Yaskawa INFORM job: DEMO_ROOF_SIDE_0625_3PAINT_16.JBI

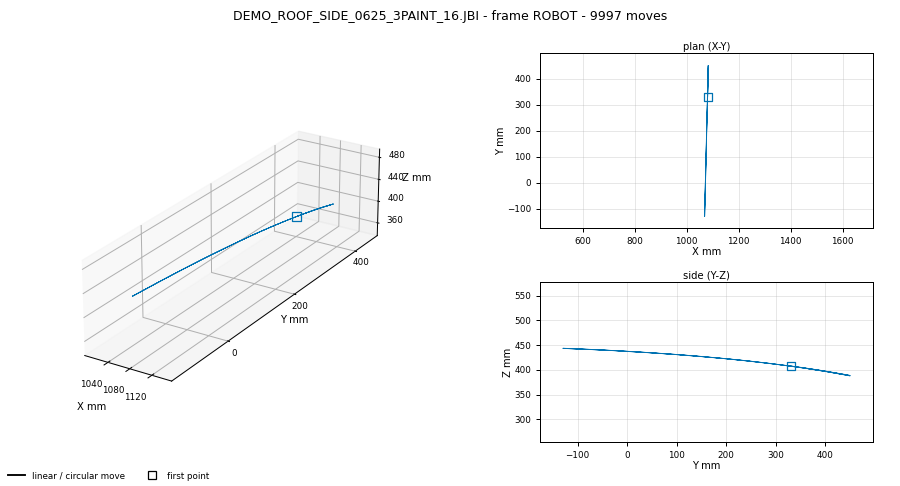
[picture p0: tool path of DEMO_ROOF_SIDE_0625_3PAINT_16.JBI in frame ROBOT, 9997 of 9997 moves have a stored position in this frame; points joined in program order, loops and branches not executed]
/JOB
//NAME DEMO_ROOF_SIDE_0625_3PAINT16
//POS
///NPOS 9997,0,0,0,0,0
///TOOL 0
///USER 0
///POSTYPE ROBOT
///RECTAN
///RCONF 1,0,0,0,0,0,0,0,0,0,0,0,0,0,0,0,0,0,0,0,0,0,0,0
C00000=1080.812,330.595,407.763,175.918,27.097,154.616
C00001=1080.821,331.010,407.707,175.923,27.105,154.617
C00002=1080.832,331.424,407.651,175.928,27.113,154.618
C00003=1080.838,331.672,407.618,175.931,27.117,154.619
C00004=1080.844,331.919,407.584,175.934,27.122,154.620
C00005=1080.849,332.167,407.551,175.937,27.126,154.620
C00006=1080.856,332.416,407.518,175.940,27.131,154.621
C00007=1080.862,332.663,407.484,175.943,27.136,154.622
C00008=1080.868,332.911,407.450,175.947,27.141,154.623
C00009=1080.873,333.158,407.416,175.950,27.146,154.623
C00010=1080.879,333.406,407.383,175.953,27.150,154.624
C00011=1080.885,333.653,407.349,175.956,27.155,154.625
C00012=1080.892,333.902,407.316,175.959,27.160,154.626
C00013=1080.898,334.149,407.282,175.962,27.165,154.627
C00014=1080.904,334.396,407.248,175.965,27.170,154.627
C00015=1080.909,334.644,407.214,175.968,27.174,154.628
C00016=1080.915,334.891,407.180,175.971,27.179,154.629
C00017=1080.921,335.140,407.147,175.975,27.183,154.630
C00018=1080.927,335.387,407.112,175.978,27.188,154.630
C00019=1080.933,335.635,407.078,175.981,27.193,154.631
C00020=1080.939,335.883,407.045,175.984,27.198,154.632
C00021=1080.946,336.130,407.011,175.987,27.202,154.633
C00022=1080.951,336.377,406.977,175.990,27.207,154.633
C00023=1080.957,336.625,406.944,175.994,27.212,154.634
C00024=1080.963,336.873,406.909,175.997,27.217,154.635
C00025=1080.969,337.121,406.875,176.000,27.222,154.636
C00026=1080.975,337.368,406.841,176.003,27.227,154.637
C00027=1080.981,337.616,406.808,176.006,27.232,154.637
C00028=1080.987,337.864,406.774,176.009,27.236,154.638
C00029=1080.993,338.111,406.740,176.012,27.241,154.639
C00030=1080.999,338.359,406.705,176.015,27.246,154.640
C00031=1081.005,338.606,406.671,176.018,27.251,154.641
C00032=1081.011,338.854,406.637,176.022,27.256,154.642
C00033=1081.018,339.102,406.603,176.025,27.261,154.642
C00034=1081.024,339.349,406.569,176.028,27.266,154.643
C00035=1081.029,339.596,406.534,176.031,27.270,154.644
C00036=1081.035,339.845,406.500,176.034,27.276,154.645
C00037=1081.041,340.092,406.466,176.037,27.280,154.646
C00038=1081.047,340.340,406.432,176.040,27.285,154.646
C00039=1081.053,340.588,406.398,176.043,27.290,154.647
C00040=1081.059,340.835,406.364,176.047,27.295,154.648
C00041=1081.065,341.082,406.329,176.050,27.300,154.649
C00042=1081.071,341.330,406.294,176.053,27.305,154.650
C00043=1081.077,341.577,406.260,176.056,27.310,154.650
C00044=1081.083,341.825,406.225,176.059,27.315,154.651
C00045=1081.089,342.072,406.191,176.062,27.320,154.652
C00046=1081.095,342.320,406.157,176.065,27.325,154.653
C00047=1081.101,342.568,406.123,176.069,27.330,154.654
C00048=1081.106,342.815,406.088,176.072,27.335,154.655
C00049=1081.113,343.063,406.054,176.075,27.340,154.655
C00050=1081.119,343.310,406.019,176.078,27.345,154.656
C00051=1081.129,343.719,405.962,176.084,27.353,154.658
C00052=1081.140,344.129,405.905,176.089,27.362,154.659
C00053=1081.149,344.538,405.848,176.095,27.370,154.660
C00054=1081.159,344.947,405.790,176.100,27.379,154.662
C00055=1081.165,345.194,405.756,176.103,27.383,154.663
C00056=1081.171,345.442,405.720,176.106,27.389,154.664
C00057=1081.177,345.689,405.686,176.109,27.394,154.665
C00058=1081.183,345.937,405.651,176.113,27.399,154.665
C00059=1081.189,346.184,405.617,176.116,27.404,154.666
C00060=1081.195,346.432,405.582,176.119,27.409,154.667
C00061=1081.201,346.679,405.547,176.122,27.414,154.668
C00062=1081.207,346.927,405.512,176.125,27.419,154.669
C00063=1081.213,347.174,405.477,176.129,27.425,154.670
C00064=1081.219,347.422,405.443,176.132,27.430,154.671
C00065=1081.225,347.669,405.407,176.135,27.435,154.671
C00066=1081.231,347.917,405.373,176.138,27.440,154.672
C00067=1081.237,348.164,405.337,176.142,27.446,154.673
C00068=1081.243,348.412,405.303,176.145,27.451,154.674
C00069=1081.250,348.659,405.268,176.148,27.456,154.675
C00070=1081.255,348.906,405.233,176.151,27.461,154.676
C00071=1081.261,349.154,405.198,176.154,27.466,154.677
C00072=1081.267,349.401,405.163,176.158,27.472,154.678
C00073=1081.273,349.649,405.127,176.161,27.477,154.679
C00074=1081.280,349.897,405.093,176.164,27.482,154.680
C00075=1081.285,350.144,405.057,176.167,27.488,154.680
C00076=1081.292,350.391,405.022,176.171,27.493,154.681
C00077=1081.298,350.639,404.987,176.174,27.498,154.682
C00078=1081.304,350.886,404.952,176.177,27.504,154.683
C00079=1081.310,351.134,404.917,176.181,27.509,154.684
C00080=1081.317,351.381,404.882,176.184,27.514,154.685
C00081=1081.322,351.628,404.846,176.187,27.519,154.686
C00082=1081.328,351.876,404.811,176.190,27.525,154.687
C00083=1081.334,352.124,404.776,176.194,27.530,154.688
C00084=1081.340,352.371,404.741,176.197,27.535,154.689
C00085=1081.347,352.618,404.706,176.200,27.541,154.689
C00086=1081.353,352.866,404.670,176.203,27.546,154.690
C00087=1081.359,353.113,404.634,176.207,27.552,154.691
C00088=1081.364,353.360,404.599,176.210,27.557,154.692
C00089=1081.371,353.608,404.564,176.213,27.562,154.693
C00090=1081.377,353.855,404.528,176.217,27.568,154.694
C00091=1081.382,354.102,404.492,176.220,27.573,154.695
C00092=1081.388,354.350,404.457,176.223,27.579,154.696
C00093=1081.395,354.597,404.422,176.227,27.584,154.697
C00094=1081.401,354.845,404.386,176.229,27.590,154.698
C00095=1081.407,355.092,404.350,176.232,27.595,154.699
C00096=1081.413,355.340,404.315,176.236,27.601,154.700
C00097=1081.419,355.587,404.279,176.239,27.606,154.701
C00098=1081.425,355.835,404.244,176.242,27.612,154.702
C00099=1081.431,356.081,404.208,176.246,27.617,154.703
C00100=1081.437,356.329,404.172,176.249,27.622,154.704
C00101=1081.443,356.576,404.136,176.252,27.628,154.705
C00102=1081.449,356.824,404.101,176.256,27.634,154.706
C00103=1081.459,357.236,404.041,176.261,27.643,154.707
C00104=1081.470,357.647,403.981,176.267,27.652,154.709
C00105=1081.480,358.060,403.922,176.272,27.661,154.711
C00106=1081.490,358.472,403.862,176.278,27.671,154.712
C00107=1081.496,358.720,403.826,176.281,27.676,154.713
C00108=1081.503,358.967,403.790,176.284,27.682,154.714
C00109=1081.509,359.214,403.755,176.288,27.688,154.715
C00110=1081.515,359.461,403.719,176.291,27.693,154.716
C00111=1081.521,359.708,403.683,176.294,27.699,154.717
C00112=1081.527,359.955,403.647,176.298,27.705,154.718
C00113=1081.533,360.203,403.611,176.301,27.711,154.719
C00114=1081.540,360.450,403.574,176.305,27.717,154.720
C00115=1081.546,360.698,403.539,176.308,27.722,154.721
C00116=1081.552,360.945,403.502,176.311,27.727,154.722
C00117=1081.558,361.193,403.467,176.315,27.733,154.723
C00118=1081.564,361.440,403.430,176.318,27.739,154.724
C00119=1081.570,361.688,403.394,176.322,27.745,154.725
C00120=1081.576,361.935,403.357,176.324,27.751,154.726
C00121=1081.582,362.181,403.321,176.327,27.756,154.727
C00122=1081.588,362.429,403.286,176.331,27.762,154.728
C00123=1081.594,362.676,403.249,176.334,27.768,154.729
C00124=1081.601,362.923,403.213,176.338,27.774,154.730
C00125=1081.607,363.170,403.177,176.341,27.780,154.731
C00126=1081.613,363.417,403.140,176.344,27.785,154.733
C00127=1081.619,363.665,403.104,176.348,27.792,154.734
C00128=1081.626,363.912,403.068,176.351,27.797,154.735
C00129=1081.631,364.160,403.031,176.355,27.803,154.736
C00130=1081.637,364.407,402.995,176.358,27.809,154.737
C00131=1081.644,364.654,402.958,176.362,27.815,154.738
C00132=1081.650,364.901,402.922,176.365,27.821,154.739
C00133=1081.657,365.148,402.885,176.369,27.827,154.740
C00134=1081.663,365.396,402.849,176.372,27.833,154.741
C00135=1081.669,365.643,402.812,176.374,27.839,154.742
C00136=1081.675,365.891,402.776,176.378,27.845,154.743
C00137=1081.681,366.138,402.739,176.381,27.850,154.744
C00138=1081.687,366.385,402.702,176.385,27.857,154.745
C00139=1081.693,366.632,402.666,176.388,27.862,154.746
C00140=1081.699,366.879,402.629,176.392,27.869,154.748
C00141=1081.705,367.126,402.592,176.395,27.875,154.749
C00142=1081.712,367.373,402.555,176.399,27.881,154.750
C00143=1081.717,367.620,402.518,176.402,27.887,154.751
C00144=1081.724,367.867,402.482,176.406,27.893,154.752
C00145=1081.730,368.114,402.445,176.409,27.899,154.753
C00146=1081.736,368.362,402.408,176.412,27.906,154.754
C00147=1081.742,368.609,402.372,176.415,27.911,154.755
C00148=1081.748,368.857,402.334,176.419,27.918,154.756
C00149=1081.755,369.103,402.297,176.422,27.924,154.758
C00150=1081.761,369.350,402.261,176.426,27.930,154.759
C00151=1081.767,369.598,402.224,176.429,27.936,154.760
C00152=1081.773,369.845,402.187,176.433,27.942,154.761
C00153=1081.779,370.092,402.150,176.436,27.948,154.762
C00154=1081.786,370.339,402.113,176.440,27.955,154.763
C00155=1081.791,370.553,402.081,176.443,27.960,154.764
C00156=1081.796,370.767,402.050,176.446,27.966,154.765
C00157=1081.801,370.981,402.017,176.448,27.970,154.766
C00158=1081.807,371.195,401.985,176.451,27.976,154.767
C00159=1081.812,371.409,401.953,176.454,27.981,154.768
C00160=1081.818,371.623,401.920,176.457,27.987,154.769
C00161=1081.823,371.837,401.888,176.460,27.992,154.770
C00162=1081.828,372.052,401.856,176.463,27.998,154.771
C00163=1081.835,372.299,401.819,176.467,28.004,154.772
C00164=1081.841,372.546,401.782,176.470,28.010,154.773
C00165=1081.847,372.792,401.745,176.474,28.016,154.775
C00166=1081.854,373.041,401.707,176.477,28.023,154.776
C00167=1081.860,373.287,401.670,176.480,28.030,154.777
C00168=1081.866,373.534,401.633,176.483,28.036,154.778
C00169=1081.873,373.781,401.596,176.487,28.042,154.779
C00170=1081.879,374.028,401.558,176.491,28.048,154.781
C00171=1081.885,374.276,401.521,176.494,28.055,154.782
C00172=1081.891,374.522,401.484,176.498,28.061,154.783
C00173=1081.898,374.769,401.445,176.501,28.068,154.784
C00174=1081.903,375.017,401.408,176.505,28.074,154.785
C00175=1081.909,375.264,401.371,176.508,28.081,154.787
C00176=1081.916,375.510,401.333,176.511,28.087,154.788
C00177=1081.922,375.757,401.295,176.515,28.094,154.789
C00178=1081.928,376.005,401.258,176.518,28.100,154.790
C00179=1081.934,376.252,401.221,176.522,28.107,154.792
C00180=1081.941,376.499,401.183,176.526,28.114,154.793
C00181=1081.947,376.745,401.145,176.529,28.120,154.794
C00182=1081.953,376.992,401.108,176.533,28.127,154.795
C00183=1081.960,377.240,401.069,176.535,28.133,154.797
C00184=1081.965,377.487,401.032,176.539,28.140,154.798
C00185=1081.972,377.733,400.995,176.543,28.146,154.799
C00186=1081.978,377.981,400.957,176.546,28.153,154.800
C00187=1081.984,378.228,400.919,176.550,28.160,154.802
C00188=1081.991,378.475,400.881,176.554,28.167,154.803
C00189=1081.997,378.722,400.843,176.557,28.173,154.804
C00190=1082.004,378.969,400.806,176.560,28.180,154.805
C00191=1082.010,379.216,400.768,176.564,28.187,154.807
C00192=1082.016,379.462,400.730,176.567,28.193,154.808
C00193=1082.022,379.709,400.692,176.571,28.200,154.809
C00194=1082.028,379.956,400.654,176.575,28.207,154.810
C00195=1082.035,380.203,400.616,176.578,28.214,154.812
C00196=1082.041,380.450,400.578,176.582,28.220,154.813
C00197=1082.048,380.697,400.540,176.585,28.227,154.814
C00198=1082.054,380.944,400.503,176.588,28.234,154.816
C00199=1082.061,381.191,400.464,176.592,28.241,154.817
C00200=1082.067,381.438,400.426,176.596,28.248,154.818
C00201=1082.073,381.685,400.388,176.599,28.255,154.820
C00202=1082.080,381.932,400.350,176.603,28.261,154.821
C00203=1082.086,382.179,400.311,176.606,28.268,154.822
C00204=1082.092,382.426,400.273,176.610,28.275,154.823
C00205=1082.098,382.673,400.235,176.613,28.282,154.825
C00206=1082.105,382.920,400.197,176.617,28.289,154.826
C00207=1082.111,383.166,400.159,176.621,28.296,154.827
C00208=1082.118,383.413,400.120,176.624,28.303,154.829
C00209=1082.123,383.660,400.082,176.627,28.310,154.830
C00210=1082.130,383.907,400.043,176.631,28.318,154.832
C00211=1082.136,384.135,400.007,176.634,28.324,154.833
C00212=1082.141,384.364,399.972,176.638,28.330,154.834
C00213=1082.148,384.592,399.937,176.641,28.337,154.835
C00214=1082.153,384.819,399.901,176.644,28.344,154.837
C00215=1082.159,385.048,399.865,176.648,28.350,154.838
C00216=1082.165,385.276,399.830,176.651,28.356,154.839
C00217=1082.171,385.505,399.794,176.655,28.363,154.840
C00218=1082.177,385.733,399.759,176.658,28.370,154.842
C00219=1082.182,385.980,399.720,176.661,28.377,154.843
C00220=1082.189,386.227,399.681,176.665,28.385,154.844
C00221=1082.195,386.474,399.643,176.668,28.392,154.846
C00222=1082.201,386.721,399.605,176.672,28.399,154.847
C00223=1082.208,386.967,399.566,176.676,28.406,154.849
C00224=1082.214,387.214,399.527,176.680,28.413,154.850
C00225=1082.220,387.461,399.488,176.683,28.421,154.852
C00226=1082.227,387.708,399.450,176.686,28.428,154.853
C00227=1082.234,387.955,399.411,176.690,28.435,154.854
C00228=1082.240,388.202,399.372,176.694,28.442,154.856
C00229=1082.246,388.448,399.333,176.698,28.450,154.857
C00230=1082.253,388.695,399.294,176.701,28.458,154.859
C00231=1082.260,388.942,399.256,176.705,28.465,154.860
C00232=1082.266,389.189,399.216,176.708,28.472,154.862
C00233=1082.272,389.435,399.178,176.712,28.479,154.863
C00234=1082.279,389.682,399.139,176.716,28.487,154.865
C00235=1082.285,389.929,399.099,176.719,28.494,154.866
C00236=1082.292,390.176,399.061,176.723,28.502,154.867
C00237=1082.298,390.423,399.022,176.727,28.509,154.869
C00238=1082.304,390.669,398.983,176.731,28.517,154.870
C00239=1082.311,390.916,398.944,176.734,28.524,154.872
C00240=1082.318,391.163,398.905,176.738,28.531,154.873
C00241=1082.324,391.410,398.866,176.741,28.539,154.875
C00242=1082.330,391.657,398.827,176.745,28.546,154.876
C00243=1082.338,391.903,398.787,176.749,28.554,154.878
C00244=1082.344,392.150,398.748,176.753,28.562,154.879
C00245=1082.350,392.396,398.709,176.756,28.570,154.881
C00246=1082.356,392.643,398.670,176.760,28.578,154.882
C00247=1082.362,392.890,398.630,176.763,28.585,154.884
C00248=1082.369,393.137,398.591,176.767,28.593,154.885
C00249=1082.375,393.384,398.551,176.771,28.601,154.887
C00250=1082.382,393.630,398.512,176.774,28.608,154.888
C00251=1082.388,393.877,398.472,176.778,28.616,154.890
C00252=1082.395,394.124,398.434,176.782,28.624,154.892
C00253=1082.402,394.370,398.393,176.786,28.632,154.893
C00254=1082.408,394.618,398.354,176.790,28.639,154.895
C00255=1082.415,394.864,398.314,176.793,28.647,154.896
C00256=1082.421,395.111,398.275,176.797,28.655,154.898
C00257=1082.427,395.357,398.235,176.801,28.663,154.899
C00258=1082.434,395.604,398.196,176.805,28.671,154.901
C00259=1082.440,395.851,398.156,176.808,28.679,154.903
C00260=1082.446,396.098,398.116,176.812,28.687,154.904
C00261=1082.453,396.344,398.076,176.816,28.695,154.906
C00262=1082.460,396.591,398.037,176.819,28.703,154.907
C00263=1082.466,396.838,397.997,176.823,28.711,154.909
C00264=1082.472,397.084,397.957,176.826,28.719,154.911
C00265=1082.479,397.331,397.918,176.830,28.727,154.912
C00266=1082.486,397.578,397.878,176.834,28.735,154.914
C00267=1082.491,397.813,397.839,176.838,28.743,154.915
C00268=1082.498,398.048,397.802,176.842,28.750,154.917
C00269=1082.504,398.283,397.764,176.845,28.759,154.919
C00270=1082.510,398.519,397.725,176.848,28.766,154.920
C00271=1082.517,398.754,397.687,176.852,28.774,154.922
C00272=1082.523,398.989,397.650,176.856,28.782,154.923
C00273=1082.529,399.224,397.611,176.860,28.790,154.925
C00274=1082.536,399.461,397.573,176.863,28.798,154.926
C00275=1082.542,399.707,397.533,176.867,28.806,154.928
C00276=1082.548,399.954,397.493,176.871,28.814,154.930
C00277=1082.555,400.200,397.453,176.875,28.823,154.932
C00278=1082.561,400.447,397.413,176.878,28.831,154.933
C00279=1082.568,400.693,397.372,176.882,28.840,154.935
C00280=1082.575,400.940,397.332,176.886,28.848,154.937
C00281=1082.581,401.187,397.292,176.890,28.856,154.938
C00282=1082.587,401.433,397.252,176.893,28.865,154.940
C00283=1082.594,401.680,397.211,176.897,28.873,154.942
C00284=1082.601,401.927,397.171,176.901,28.882,154.944
C00285=1082.607,402.174,397.131,176.905,28.890,154.945
C00286=1082.614,402.420,397.090,176.908,28.898,154.947
C00287=1082.621,402.667,397.049,176.913,28.907,154.949
C00288=1082.627,402.913,397.009,176.917,28.916,154.950
C00289=1082.633,403.160,396.969,176.921,28.924,154.952
C00290=1082.641,403.406,396.928,176.924,28.933,154.954
C00291=1082.646,403.653,396.887,176.928,28.942,154.956
C00292=1082.653,403.900,396.847,176.932,28.950,154.958
C00293=1082.660,404.147,396.807,176.936,28.959,154.959
C00294=1082.666,404.393,396.766,176.939,28.968,154.961
C00295=1082.673,404.639,396.726,176.944,28.976,154.963
C00296=1082.680,404.886,396.684,176.948,28.985,154.965
C00297=1082.686,405.133,396.644,176.952,28.994,154.967
C00298=1082.692,405.379,396.603,176.955,29.002,154.968
C00299=1082.699,405.626,396.562,176.959,29.012,154.970
C00300=1082.706,405.872,396.522,176.964,29.021,154.972
C00301=1082.712,406.119,396.480,176.968,29.030,154.974
C00302=1082.719,406.365,396.439,176.971,29.038,154.976
C00303=1082.726,406.612,396.399,176.975,29.047,154.978
C00304=1082.733,406.858,396.358,176.979,29.056,154.980
C00305=1082.738,407.105,396.317,176.983,29.065,154.981
C00306=1082.746,407.352,396.276,176.987,29.074,154.983
C00307=1082.752,407.598,396.235,176.991,29.083,154.985
C00308=1082.759,407.845,396.193,176.995,29.092,154.987
C00309=1082.765,408.091,396.153,176.999,29.102,154.989
C00310=1082.772,408.338,396.111,177.003,29.111,154.991
C00311=1082.778,408.584,396.070,177.007,29.120,154.993
C00312=1082.785,408.831,396.029,177.011,29.129,154.995
C00313=1082.791,409.077,395.988,177.015,29.139,154.997
C00314=1082.798,409.324,395.947,177.019,29.148,154.999
C00315=1082.805,409.570,395.906,177.023,29.157,155.001
C00316=1082.811,409.817,395.864,177.027,29.167,155.003
C00317=1082.818,410.064,395.823,177.031,29.176,155.004
C00318=1082.824,410.310,395.781,177.035,29.185,155.006
C00319=1082.832,410.556,395.740,177.040,29.195,155.008
C00320=1082.838,410.803,395.699,177.043,29.204,155.010
C00321=1082.845,411.049,395.657,177.047,29.213,155.012
C00322=1082.851,411.296,395.616,177.052,29.223,155.014
C00323=1082.858,411.532,395.576,177.056,29.232,155.016
C00324=1082.864,411.768,395.536,177.059,29.241,155.018
C00325=1082.871,412.005,395.496,177.063,29.250,155.020
C00326=1082.877,412.241,395.456,177.067,29.260,155.022
C00327=1082.884,412.477,395.417,177.072,29.269,155.024
C00328=1082.891,412.713,395.376,177.075,29.278,155.026
C00329=1082.897,412.949,395.337,177.079,29.287,155.028
C00330=1082.903,413.186,395.297,177.083,29.296,155.030
C00331=1082.910,413.432,395.254,177.088,29.306,155.032
C00332=1082.917,413.678,395.213,177.091,29.316,155.034
C00333=1082.923,413.925,395.172,177.096,29.326,155.036
C00334=1082.931,414.171,395.130,177.100,29.335,155.038
C00335=1082.937,414.418,395.088,177.104,29.345,155.040
C00336=1082.944,414.664,395.045,177.108,29.355,155.042
C00337=1082.951,414.910,395.005,177.112,29.365,155.044
C00338=1082.958,415.156,394.962,177.117,29.375,155.046
C00339=1082.964,415.403,394.920,177.120,29.384,155.048
C00340=1082.972,415.649,394.878,177.125,29.394,155.051
C00341=1082.979,415.896,394.836,177.129,29.404,155.053
C00342=1082.985,416.142,394.794,177.134,29.414,155.055
C00343=1082.992,416.389,394.752,177.137,29.424,155.057
C00344=1082.998,416.635,394.710,177.142,29.435,155.059
C00345=1083.005,416.881,394.667,177.147,29.445,155.061
C00346=1083.013,417.127,394.625,177.150,29.455,155.063
C00347=1083.019,417.374,394.584,177.155,29.465,155.066
C00348=1083.026,417.620,394.541,177.159,29.476,155.068
C00349=1083.033,417.867,394.498,177.163,29.486,155.070
C00350=1083.040,418.113,394.456,177.167,29.496,155.072
C00351=1083.046,418.359,394.414,177.172,29.506,155.074
C00352=1083.053,418.605,394.371,177.177,29.517,155.077
C00353=1083.060,418.851,394.329,177.180,29.527,155.079
C00354=1083.066,419.098,394.287,177.185,29.538,155.081
C00355=1083.073,419.344,394.244,177.190,29.548,155.083
C00356=1083.080,419.591,394.202,177.193,29.558,155.086
C00357=1083.087,419.836,394.158,177.198,29.569,155.088
C00358=1083.094,420.083,394.116,177.202,29.580,155.090
C00359=1083.101,420.329,394.073,177.207,29.590,155.092
C00360=1083.108,420.575,394.031,177.211,29.600,155.095
C00361=1083.115,420.821,393.988,177.215,29.611,155.097
C00362=1083.121,421.068,393.946,177.220,29.622,155.099
C00363=1083.129,421.315,393.903,177.224,29.632,155.102
C00364=1083.136,421.560,393.860,177.229,29.644,155.104
C00365=1083.143,421.807,393.817,177.233,29.654,155.106
C00366=1083.150,422.053,393.775,177.238,29.665,155.109
C00367=1083.157,422.299,393.731,177.242,29.676,155.111
C00368=1083.164,422.545,393.689,177.247,29.687,155.113
C00369=1083.171,422.791,393.646,177.251,29.698,155.116
C00370=1083.177,423.037,393.602,177.255,29.708,155.118
C00371=1083.184,423.283,393.560,177.260,29.719,155.120
C00372=1083.191,423.529,393.517,177.265,29.731,155.123
C00373=1083.199,423.776,393.474,177.268,29.741,155.125
C00374=1083.205,424.022,393.430,177.273,29.753,155.128
C00375=1083.212,424.268,393.387,177.278,29.764,155.130
C00376=1083.219,424.514,393.344,177.283,29.775,155.133
C00377=1083.225,424.760,393.300,177.287,29.786,155.135
C00378=1083.233,425.007,393.257,177.291,29.797,155.138
C00379=1083.240,425.254,393.213,177.296,29.809,155.140
C00380=1083.247,425.501,393.170,177.300,29.820,155.142
C00381=1083.254,425.748,393.127,177.305,29.831,155.145
C00382=1083.261,425.995,393.083,177.310,29.843,155.147
C00383=1083.268,426.241,393.040,177.315,29.854,155.150
C00384=1083.275,426.487,392.997,177.319,29.866,155.152
C00385=1083.282,426.733,392.952,177.324,29.877,155.155
C00386=1083.289,426.979,392.909,177.329,29.888,155.157
C00387=1083.296,427.225,392.866,177.332,29.900,155.160
C00388=1083.304,427.471,392.822,177.337,29.911,155.163
C00389=1083.311,427.717,392.778,177.342,29.923,155.165
C00390=1083.317,427.963,392.735,177.347,29.935,155.168
C00391=1083.325,428.209,392.691,177.351,29.947,155.170
C00392=1083.332,428.455,392.648,177.356,29.958,155.173
C00393=1083.339,428.702,392.603,177.361,29.970,155.175
C00394=1083.345,428.948,392.560,177.366,29.982,155.178
C00395=1083.353,429.193,392.516,177.370,29.994,155.181
C00396=1083.360,429.439,392.471,177.375,30.006,155.183
C00397=1083.367,429.685,392.428,177.380,30.018,155.186
C00398=1083.374,429.932,392.384,177.384,30.030,155.189
C00399=1083.382,430.177,392.340,177.389,30.042,155.191
C00400=1083.388,430.423,392.296,177.394,30.054,155.194
C00401=1083.395,430.669,392.251,177.399,30.066,155.197
C00402=1083.403,430.914,392.208,177.403,30.078,155.199
C00403=1083.410,431.160,392.163,177.408,30.090,155.202
C00404=1083.417,431.406,392.120,177.413,30.102,155.205
C00405=1083.424,431.652,392.075,177.418,30.114,155.208
C00406=1083.431,431.899,392.031,177.423,30.127,155.210
C00407=1083.439,432.144,391.987,177.428,30.139,155.213
C00408=1083.446,432.391,391.942,177.433,30.152,155.216
C00409=1083.453,432.636,391.898,177.438,30.164,155.218
C00410=1083.460,432.882,391.853,177.442,30.176,155.221
C00411=1083.466,433.128,391.809,177.447,30.189,155.224
C00412=1083.474,433.374,391.765,177.452,30.202,155.227
C00413=1083.482,433.620,391.720,177.457,30.214,155.230
C00414=1083.489,433.865,391.675,177.462,30.227,155.233
C00415=1083.496,434.111,391.630,177.467,30.239,155.235
C00416=1083.503,434.356,391.586,177.472,30.252,155.238
C00417=1083.510,434.602,391.541,177.477,30.265,155.241
C00418=1083.517,434.849,391.496,177.481,30.278,155.244
C00419=1083.524,435.092,391.452,177.486,30.291,155.247
C00420=1083.531,435.335,391.408,177.492,30.303,155.250
C00421=1083.538,435.579,391.363,177.497,30.316,155.253
C00422=1083.545,435.823,391.319,177.501,30.329,155.256
C00423=1083.553,436.066,391.274,177.506,30.342,155.259
C00424=1083.560,436.309,391.230,177.511,30.355,155.261
C00425=1083.567,436.553,391.185,177.517,30.368,155.264
C00426=1083.575,436.796,391.140,177.522,30.381,155.267
C00427=1083.582,437.042,391.095,177.526,30.394,155.270
C00428=1083.589,437.288,391.050,177.531,30.407,155.273
C00429=1083.596,437.533,391.005,177.537,30.421,155.276
C00430=1083.604,437.779,390.960,177.542,30.434,155.279
C00431=1083.611,438.025,390.915,177.547,30.447,155.283
C00432=1083.619,438.270,390.870,177.552,30.460,155.285
C00433=1083.626,438.517,390.825,177.557,30.474,155.289
C00434=1083.634,438.762,390.779,177.563,30.487,155.292
C00435=1083.644,439.107,390.716,177.569,30.507,155.296
C00436=1083.655,439.451,390.652,177.577,30.525,155.300
C00437=1083.665,439.796,390.588,177.584,30.545,155.305
C00438=1083.676,440.141,390.524,177.591,30.564,155.309
C00439=1083.683,440.386,390.479,177.597,30.578,155.312
C00440=1083.690,440.631,390.433,177.602,30.592,155.315
C00441=1083.697,440.877,390.388,177.608,30.606,155.319
C00442=1083.704,441.123,390.342,177.613,30.620,155.322
C00443=1083.712,441.368,390.296,177.618,30.634,155.325
C00444=1083.720,441.614,390.250,177.623,30.648,155.328
C00445=1083.727,441.860,390.204,177.629,30.662,155.332
C00446=1083.735,442.106,390.159,177.634,30.676,155.335
C00447=1083.743,442.351,390.113,177.640,30.691,155.338
C00448=1083.749,442.597,390.067,177.645,30.705,155.342
C00449=1083.757,442.842,390.020,177.650,30.719,155.345
C00450=1083.764,443.087,389.974,177.655,30.733,155.348
C00451=1083.772,443.333,389.928,177.661,30.748,155.351
C00452=1083.780,443.578,389.883,177.667,30.763,155.355
C00453=1083.786,443.824,389.837,177.672,30.777,155.358
C00454=1083.795,444.069,389.790,177.678,30.792,155.362
C00455=1083.802,444.315,389.744,177.683,30.806,155.365
C00456=1083.810,444.560,389.697,177.689,30.821,155.368
C00457=1083.817,444.805,389.652,177.694,30.836,155.372
C00458=1083.825,445.052,389.605,177.699,30.851,155.375
C00459=1083.833,445.297,389.559,177.705,30.866,155.379
C00460=1083.840,445.542,389.512,177.711,30.881,155.382
C00461=1083.847,445.788,389.465,177.716,30.895,155.386
C00462=1083.856,446.033,389.419,177.721,30.910,155.389
C00463=1083.862,446.279,389.372,177.725,30.925,155.393
C00464=1083.870,446.524,389.326,177.730,30.940,155.396
C00465=1083.878,446.769,389.279,177.734,30.955,155.400
C00466=1083.885,447.015,389.232,177.738,30.969,155.403
C00467=1083.893,447.260,389.186,177.742,30.984,155.407
C00468=1083.901,447.506,389.139,177.746,30.999,155.410
C00469=1083.909,447.751,389.092,177.749,31.014,155.414
C00470=1083.917,447.996,389.045,177.752,31.028,155.418
C00471=1083.924,448.242,388.998,177.755,31.044,155.421
C00472=1083.932,448.486,388.952,177.758,31.058,155.425
C00473=1083.940,448.732,388.904,177.760,31.073,155.428
C00474=1083.947,448.977,388.857,177.763,31.088,155.432
C00475=1083.955,449.222,388.811,177.765,31.102,155.436
C00476=1083.963,449.468,388.764,177.767,31.117,155.439
C00477=1083.973,449.712,388.719,177.770,31.130,155.443
C00478=1083.985,449.959,388.674,177.772,31.143,155.446
C00479=1083.614,449.951,388.464,177.739,31.321,155.494
C00480=1083.601,449.705,388.508,177.737,31.309,155.490
C00481=1083.591,449.459,388.554,177.735,31.295,155.487
C00482=1083.583,449.215,388.600,177.733,31.281,155.483
C00483=1083.575,448.969,388.647,177.730,31.266,155.480
C00484=1083.567,448.725,388.694,177.728,31.251,155.476
C00485=1083.559,448.479,388.742,177.725,31.236,155.473
C00486=1083.552,448.234,388.789,177.722,31.222,155.469
C00487=1083.544,447.989,388.835,177.719,31.207,155.465
C00488=1083.536,447.744,388.882,177.716,31.192,155.462
C00489=1083.529,447.497,388.929,177.712,31.177,155.458
C00490=1083.521,447.252,388.975,177.708,31.162,155.454
C00491=1083.513,447.007,389.023,177.704,31.147,155.451
C00492=1083.506,446.761,389.070,177.700,31.132,155.447
C00493=1083.497,446.516,389.116,177.696,31.118,155.444
C00494=1083.490,446.271,389.163,177.691,31.103,155.440
C00495=1083.483,446.025,389.209,177.687,31.088,155.437
C00496=1083.475,445.780,389.256,177.682,31.073,155.433
C00497=1083.468,445.534,389.303,177.676,31.058,155.430
C00498=1083.460,445.289,389.349,177.671,31.044,155.426
C00499=1083.453,445.044,389.396,177.665,31.028,155.423
C00500=1083.444,444.798,389.443,177.660,31.014,155.419
C00501=1083.437,444.553,389.489,177.654,30.999,155.416
C00502=1083.429,444.308,389.535,177.648,30.984,155.412
C00503=1083.421,444.062,389.581,177.643,30.969,155.409
C00504=1083.414,443.816,389.627,177.637,30.955,155.406
C00505=1083.406,443.571,389.674,177.631,30.940,155.402
C00506=1083.399,443.325,389.720,177.626,30.926,155.399
C00507=1083.392,443.080,389.766,177.620,30.911,155.396
C00508=1083.384,442.834,389.813,177.615,30.897,155.392
C00509=1083.376,442.589,389.859,177.609,30.883,155.389
C00510=1083.369,442.343,389.904,177.604,30.868,155.386
C00511=1083.362,442.098,389.951,177.598,30.854,155.382
C00512=1083.354,441.852,389.996,177.593,30.840,155.379
C00513=1083.346,441.607,390.042,177.587,30.826,155.376
C00514=1083.340,441.361,390.088,177.582,30.811,155.372
C00515=1083.332,441.116,390.134,177.577,30.797,155.369
C00516=1083.324,440.870,390.179,177.572,30.784,155.366
C00517=1083.317,440.625,390.225,177.566,30.770,155.363
C00518=1083.310,440.379,390.271,177.561,30.756,155.360
C00519=1083.302,440.133,390.317,177.555,30.742,155.357
C00520=1083.292,439.804,390.378,177.548,30.723,155.352
C00521=1083.282,439.474,390.439,177.541,30.705,155.348
C00522=1083.272,439.145,390.500,177.534,30.687,155.344
C00523=1083.262,438.816,390.560,177.527,30.668,155.340
C00524=1083.254,438.571,390.606,177.522,30.655,155.337
C00525=1083.247,438.325,390.652,177.516,30.641,155.334
C00526=1083.239,438.079,390.697,177.511,30.628,155.331
C00527=1083.232,437.834,390.742,177.506,30.615,155.327
C00528=1083.224,437.588,390.787,177.500,30.601,155.324
C00529=1083.217,437.342,390.832,177.495,30.588,155.321
C00530=1083.209,437.096,390.878,177.491,30.575,155.318
C00531=1083.202,436.850,390.923,177.485,30.561,155.315
C00532=1083.195,436.606,390.968,177.480,30.548,155.312
C00533=1083.188,436.359,391.013,177.475,30.535,155.309
C00534=1083.180,436.113,391.058,177.470,30.522,155.306
C00535=1083.173,435.867,391.103,177.464,30.509,155.303
C00536=1083.165,435.622,391.148,177.459,30.496,155.301
C00537=1083.159,435.377,391.193,177.454,30.483,155.298
C00538=1083.151,435.131,391.238,177.450,30.470,155.295
C00539=1083.144,434.884,391.283,177.444,30.457,155.292
C00540=1083.137,434.639,391.327,177.439,30.445,155.289
C00541=1083.130,434.393,391.372,177.434,30.432,155.286
C00542=1083.123,434.147,391.417,177.429,30.419,155.283
C00543=1083.116,433.902,391.462,177.424,30.406,155.280
C00544=1083.108,433.656,391.506,177.420,30.394,155.277
C00545=1083.100,433.410,391.551,177.414,30.381,155.275
C00546=1083.094,433.164,391.596,177.409,30.368,155.272
C00547=1083.087,432.918,391.640,177.404,30.356,155.269
C00548=1083.080,432.672,391.685,177.399,30.343,155.266
C00549=1083.073,432.426,391.729,177.394,30.331,155.263
C00550=1083.065,432.181,391.774,177.390,30.318,155.261
C00551=1083.058,431.935,391.818,177.385,30.306,155.258
C00552=1083.051,431.689,391.863,177.380,30.294,155.255
C00553=1083.043,431.443,391.907,177.375,30.282,155.252
C00554=1083.036,431.197,391.951,177.370,30.269,155.250
C00555=1083.029,430.951,391.996,177.365,30.257,155.247
C00556=1083.022,430.705,392.039,177.360,30.245,155.244
C00557=1083.014,430.459,392.084,177.355,30.233,155.242
C00558=1083.008,430.213,392.128,177.350,30.221,155.239
C00559=1083.000,429.967,392.172,177.345,30.209,155.236
C00560=1082.994,429.721,392.216,177.340,30.197,155.233
C00561=1082.986,429.475,392.260,177.336,30.185,155.231
C00562=1082.979,429.230,392.304,177.331,30.173,155.228
C00563=1082.972,428.984,392.347,177.326,30.161,155.225
C00564=1082.965,428.737,392.392,177.321,30.149,155.223
C00565=1082.958,428.491,392.435,177.317,30.137,155.220
C00566=1082.951,428.245,392.479,177.313,30.126,155.218
C00567=1082.944,428.000,392.524,177.308,30.114,155.215
C00568=1082.936,427.753,392.567,177.303,30.102,155.212
C00569=1082.929,427.508,392.610,177.298,30.090,155.210
C00570=1082.923,427.262,392.654,177.293,30.079,155.207
C00571=1082.915,427.015,392.698,177.289,30.067,155.205
C00572=1082.908,426.770,392.741,177.284,30.056,155.202
C00573=1082.901,426.525,392.785,177.279,30.044,155.200
C00574=1082.894,426.280,392.828,177.274,30.033,155.197
C00575=1082.887,426.035,392.872,177.270,30.022,155.195
C00576=1082.880,425.790,392.915,177.266,30.010,155.192
C00577=1082.873,425.546,392.958,177.261,29.999,155.190
C00578=1082.865,425.301,393.001,177.256,29.988,155.187
C00579=1082.859,425.056,393.044,177.251,29.977,155.185
C00580=1082.852,424.810,393.088,177.246,29.965,155.182
C00581=1082.845,424.563,393.131,177.243,29.954,155.180
C00582=1082.838,424.317,393.174,177.238,29.943,155.177
C00583=1082.831,424.072,393.217,177.233,29.932,155.175
C00584=1082.824,423.826,393.261,177.228,29.921,155.173
C00585=1082.817,423.579,393.303,177.223,29.909,155.170
C00586=1082.810,423.333,393.347,177.220,29.899,155.168
C00587=1082.803,423.087,393.390,177.215,29.887,155.165
C00588=1082.796,422.841,393.433,177.210,29.876,155.163
C00589=1082.789,422.594,393.476,177.205,29.866,155.161
C00590=1082.782,422.349,393.519,177.202,29.855,155.158
C00591=1082.775,422.102,393.562,177.197,29.843,155.156
C00592=1082.764,421.711,393.631,177.190,29.827,155.152
C00593=1082.753,421.319,393.698,177.183,29.809,155.148
C00594=1082.742,420.927,393.766,177.176,29.793,155.145
C00595=1082.731,420.536,393.835,177.169,29.775,155.141
C00596=1082.724,420.289,393.877,177.164,29.765,155.139
C00597=1082.717,420.043,393.920,177.159,29.754,155.136
C00598=1082.710,419.797,393.962,177.155,29.744,155.134
C00599=1082.703,419.551,394.005,177.150,29.733,155.132
C00600=1082.696,419.304,394.047,177.147,29.723,155.130
C00601=1082.690,419.058,394.090,177.142,29.712,155.127
C00602=1082.683,418.812,394.132,177.137,29.702,155.125
C00603=1082.676,418.565,394.175,177.133,29.691,155.123
C00604=1082.669,418.319,394.218,177.129,29.681,155.121
C00605=1082.662,418.073,394.260,177.124,29.670,155.118
C00606=1082.655,417.827,394.303,177.120,29.660,155.116
C00607=1082.648,417.580,394.345,177.115,29.650,155.114
C00608=1082.642,417.334,394.388,177.111,29.640,155.112
C00609=1082.635,417.088,394.430,177.107,29.629,155.110
C00610=1082.628,416.842,394.471,177.103,29.619,155.108
C00611=1082.621,416.596,394.514,177.098,29.609,155.105
C00612=1082.614,416.349,394.556,177.094,29.599,155.103
C00613=1082.607,416.103,394.599,177.090,29.589,155.101
C00614=1082.601,415.856,394.641,177.086,29.579,155.099
C00615=1082.594,415.610,394.683,177.081,29.569,155.097
C00616=1082.586,415.364,394.725,177.077,29.559,155.095
C00617=1082.581,415.118,394.767,177.072,29.549,155.093
C00618=1082.574,414.871,394.809,177.069,29.539,155.090
C00619=1082.566,414.625,394.850,177.064,29.530,155.088
C00620=1082.560,414.378,394.893,177.060,29.519,155.086
C00621=1082.553,414.132,394.935,177.055,29.510,155.084
C00622=1082.545,413.886,394.977,177.052,29.500,155.082
C00623=1082.539,413.639,395.018,177.047,29.490,155.080
C00624=1082.532,413.393,395.059,177.043,29.481,155.078
C00625=1082.525,413.147,395.102,177.039,29.471,155.076
C00626=1082.519,412.900,395.144,177.034,29.461,155.074
C00627=1082.512,412.654,395.185,177.031,29.452,155.072
C00628=1082.503,412.325,395.241,177.025,29.439,155.069
C00629=1082.494,411.997,395.296,177.019,29.426,155.067
C00630=1082.484,411.669,395.352,177.014,29.413,155.064
C00631=1082.476,411.340,395.407,177.008,29.401,155.061
C00632=1082.469,411.093,395.449,177.004,29.391,155.059
C00633=1082.462,410.848,395.489,177.000,29.382,155.057
C00634=1082.456,410.601,395.531,176.996,29.372,155.055
C00635=1082.449,410.355,395.572,176.992,29.363,155.053
C00636=1082.442,410.108,395.615,176.987,29.353,155.051
C00637=1082.435,409.862,395.656,176.983,29.344,155.049
C00638=1082.429,409.616,395.697,176.980,29.335,155.047
C00639=1082.422,409.368,395.738,176.975,29.325,155.045
C00640=1082.416,409.122,395.779,176.971,29.316,155.043
C00641=1082.409,408.876,395.820,176.967,29.307,155.041
C00642=1082.403,408.629,395.862,176.964,29.298,155.040
C00643=1082.396,408.383,395.903,176.959,29.288,155.038
C00644=1082.389,408.137,395.944,176.955,29.279,155.036
C00645=1082.382,407.890,395.986,176.951,29.270,155.034
C00646=1082.376,407.644,396.026,176.947,29.261,155.032
C00647=1082.370,407.397,396.068,176.943,29.252,155.030
C00648=1082.363,407.151,396.109,176.939,29.243,155.028
C00649=1082.356,406.904,396.150,176.935,29.234,155.026
C00650=1082.350,406.657,396.191,176.931,29.225,155.024
C00651=1082.343,406.411,396.232,176.928,29.216,155.022
C00652=1082.336,406.164,396.272,176.923,29.206,155.020
C00653=1082.330,405.917,396.314,176.919,29.198,155.019
C00654=1082.323,405.671,396.355,176.915,29.189,155.017
C00655=1082.316,405.424,396.395,176.911,29.180,155.015
C00656=1082.309,405.178,396.436,176.908,29.171,155.013
C00657=1082.303,404.931,396.477,176.903,29.162,155.011
C00658=1082.296,404.685,396.518,176.899,29.153,155.010
C00659=1082.290,404.438,396.558,176.895,29.145,155.008
C00660=1082.283,404.191,396.599,176.891,29.136,155.006
C00661=1082.276,403.945,396.640,176.888,29.127,155.004
C00662=1082.270,403.698,396.681,176.884,29.119,155.002
C00663=1082.264,403.451,396.721,176.880,29.110,155.001
C00664=1082.257,403.205,396.762,176.875,29.101,154.999
C00665=1082.250,402.958,396.802,176.871,29.092,154.997
C00666=1082.244,402.712,396.842,176.868,29.084,154.995
C00667=1082.237,402.466,396.883,176.864,29.076,154.994
C00668=1082.230,402.218,396.924,176.860,29.067,154.992
C00669=1082.224,401.972,396.964,176.856,29.058,154.990
C00670=1082.217,401.725,397.004,176.852,29.050,154.988
C00671=1082.211,401.479,397.044,176.849,29.041,154.986
C00672=1082.204,401.232,397.085,176.845,29.033,154.985
C00673=1082.198,400.985,397.125,176.841,29.025,154.983
C00674=1082.191,400.739,397.166,176.837,29.016,154.981
C00675=1082.184,400.493,397.206,176.833,29.008,154.980
C00676=1082.177,400.246,397.246,176.830,28.999,154.978
C00677=1082.171,399.999,397.287,176.826,28.991,154.976
C00678=1082.165,399.753,397.327,176.822,28.983,154.974
C00679=1082.158,399.506,397.367,176.817,28.974,154.973
C00680=1082.152,399.270,397.405,176.814,28.966,154.971
C00681=1082.145,399.034,397.443,176.810,28.958,154.970
C00682=1082.140,398.798,397.481,176.807,28.951,154.968
C00683=1082.134,398.562,397.520,176.803,28.943,154.966
C00684=1082.127,398.326,397.558,176.800,28.935,154.965
C00685=1082.121,398.090,397.596,176.796,28.927,154.963
C00686=1082.114,397.854,397.634,176.792,28.919,154.962
C00687=1082.108,397.618,397.673,176.788,28.911,154.960
C00688=1082.102,397.371,397.712,176.784,28.903,154.958
C00689=1082.095,397.125,397.752,176.781,28.895,154.957
C00690=1082.088,396.878,397.792,176.777,28.887,154.955
C00691=1082.082,396.631,397.832,176.773,28.879,154.954
C00692=1082.076,396.385,397.872,176.769,28.871,154.952
C00693=1082.069,396.139,397.911,176.766,28.863,154.950
C00694=1082.063,395.891,397.951,176.762,28.855,154.949
C00695=1082.056,395.645,397.991,176.759,28.847,154.947
C00696=1082.050,395.398,398.030,176.755,28.839,154.945
C00697=1082.043,395.152,398.070,176.751,28.831,154.944
C00698=1082.037,394.905,398.110,176.747,28.823,154.942
C00699=1082.031,394.658,398.149,176.743,28.816,154.941
C00700=1082.024,394.411,398.188,176.739,28.808,154.939
C00701=1082.018,394.165,398.228,176.736,28.800,154.938
C00702=1082.012,393.918,398.268,176.732,28.792,154.936
C00703=1082.004,393.671,398.307,176.728,28.784,154.934
C00704=1081.998,393.424,398.347,176.724,28.776,154.933
C00705=1081.991,393.178,398.386,176.721,28.769,154.931
C00706=1081.985,392.931,398.426,176.717,28.761,154.930
C00707=1081.978,392.684,398.465,176.714,28.753,154.928
C00708=1081.972,392.437,398.504,176.710,28.746,154.927
C00709=1081.965,392.191,398.544,176.706,28.738,154.925
C00710=1081.959,391.944,398.583,176.702,28.730,154.924
C00711=1081.954,391.697,398.622,176.698,28.723,154.922
C00712=1081.947,391.450,398.661,176.694,28.715,154.921
C00713=1081.940,391.204,398.701,176.692,28.707,154.919
C00714=1081.934,390.957,398.740,176.688,28.700,154.918
C00715=1081.927,390.710,398.779,176.684,28.692,154.916
C00716=1081.920,390.463,398.818,176.680,28.685,154.915
C00717=1081.914,390.216,398.857,176.676,28.677,154.913
C00718=1081.907,389.969,398.896,176.672,28.670,154.912
C00719=1081.901,389.723,398.934,176.669,28.662,154.910
C00720=1081.895,389.476,398.974,176.666,28.655,154.909
C00721=1081.888,389.229,399.013,176.662,28.648,154.907
C00722=1081.881,388.982,399.051,176.658,28.640,154.906
C00723=1081.874,388.736,399.090,176.654,28.633,154.905
C00724=1081.869,388.489,399.129,176.650,28.625,154.903
C00725=1081.862,388.242,399.168,176.646,28.618,154.902
C00726=1081.855,387.996,399.207,176.644,28.611,154.900
C00727=1081.849,387.748,399.246,176.640,28.604,154.899
C00728=1081.843,387.502,399.285,176.636,28.596,154.897
C00729=1081.836,387.255,399.323,176.632,28.589,154.896
C00730=1081.830,387.008,399.362,176.628,28.581,154.895
C00731=1081.823,386.762,399.400,176.625,28.574,154.893
C00732=1081.817,386.515,399.440,176.621,28.567,154.892
C00733=1081.811,386.268,399.479,176.618,28.560,154.890
C00734=1081.805,386.021,399.516,176.614,28.552,154.889
C00735=1081.798,385.774,399.555,176.611,28.546,154.888
C00736=1081.792,385.545,399.592,176.607,28.539,154.886
C00737=1081.786,385.317,399.627,176.604,28.532,154.885
C00738=1081.780,385.087,399.663,176.600,28.526,154.884
C00739=1081.775,384.859,399.698,176.597,28.519,154.882
C00740=1081.768,384.630,399.734,176.594,28.513,154.881
C00741=1081.762,384.402,399.770,176.590,28.506,154.880
C00742=1081.757,384.172,399.806,176.587,28.499,154.879
C00743=1081.751,383.943,399.841,176.583,28.492,154.877
C00744=1081.745,383.696,399.880,176.580,28.485,154.876
C00745=1081.739,383.450,399.918,176.576,28.478,154.875
C00746=1081.732,383.203,399.957,176.573,28.471,154.873
C00747=1081.726,382.956,399.995,176.570,28.465,154.872
C00748=1081.720,382.708,400.033,176.566,28.457,154.870
C00749=1081.714,382.462,400.072,176.562,28.450,154.869
C00750=1081.707,382.215,400.110,176.558,28.443,154.868
C00751=1081.701,381.969,400.148,176.555,28.437,154.866
C00752=1081.695,381.721,400.186,176.551,28.429,154.865
C00753=1081.689,381.475,400.224,176.547,28.422,154.864
C00754=1081.682,381.227,400.262,176.545,28.416,154.862
C00755=1081.675,380.981,400.300,176.541,28.409,154.861
C00756=1081.669,380.734,400.338,176.537,28.402,154.860
C00757=1081.662,380.486,400.376,176.534,28.396,154.859
C00758=1081.656,380.240,400.414,176.530,28.388,154.857
C00759=1081.650,379.993,400.453,176.526,28.381,154.856
C00760=1081.644,379.746,400.491,176.523,28.375,154.855
C00761=1081.637,379.499,400.529,176.519,28.368,154.853
C00762=1081.631,379.252,400.566,176.515,28.361,154.852
C00763=1081.625,379.005,400.604,176.513,28.355,154.851
C00764=1081.618,378.758,400.642,176.509,28.348,154.850
C00765=1081.612,378.511,400.680,176.505,28.341,154.848
C00766=1081.606,378.264,400.718,176.502,28.335,154.847
C00767=1081.600,378.017,400.756,176.498,28.328,154.846
C00768=1081.593,377.770,400.793,176.495,28.321,154.845
C00769=1081.587,377.523,400.831,176.491,28.315,154.843
C00770=1081.581,377.276,400.869,176.487,28.308,154.842
C00771=1081.574,377.029,400.907,176.484,28.302,154.841
C00772=1081.568,376.782,400.944,176.480,28.295,154.840
C00773=1081.561,376.535,400.982,176.478,28.288,154.838
C00774=1081.555,376.288,401.020,176.474,28.282,154.837
C00775=1081.550,376.041,401.057,176.470,28.275,154.836
C00776=1081.543,375.794,401.095,176.467,28.268,154.834
C00777=1081.537,375.547,401.133,176.463,28.262,154.833
C00778=1081.531,375.300,401.170,176.460,28.255,154.832
C00779=1081.525,375.054,401.208,176.456,28.249,154.831
C00780=1081.519,374.806,401.245,176.452,28.242,154.830
C00781=1081.513,374.559,401.283,176.449,28.236,154.828
C00782=1081.506,374.312,401.320,176.445,28.229,154.827
C00783=1081.500,374.064,401.357,176.442,28.223,154.826
C00784=1081.494,373.818,401.395,176.439,28.216,154.825
C00785=1081.487,373.571,401.432,176.436,28.210,154.824
C00786=1081.481,373.323,401.470,176.432,28.204,154.822
C00787=1081.474,373.077,401.507,176.429,28.198,154.821
C00788=1081.469,372.829,401.544,176.425,28.191,154.820
C00789=1081.462,372.582,401.581,176.421,28.184,154.819
C00790=1081.456,372.335,401.618,176.418,28.178,154.818
C00791=1081.449,372.088,401.656,176.414,28.172,154.817
C00792=1081.444,371.874,401.688,176.411,28.166,154.815
C00793=1081.438,371.659,401.720,176.408,28.161,154.815
C00794=1081.433,371.444,401.752,176.406,28.156,154.813
C00795=1081.427,371.229,401.785,176.403,28.150,154.812
C00796=1081.423,371.015,401.817,176.400,28.145,154.812
C00797=1081.417,370.800,401.849,176.397,28.139,154.810
C00798=1081.412,370.585,401.881,176.394,28.134,154.809
C00799=1081.406,370.371,401.914,176.390,28.129,154.809
C00800=1081.400,370.124,401.951,176.387,28.122,154.807
C00801=1081.394,369.877,401.988,176.384,28.116,154.806
C00802=1081.388,369.630,402.024,176.380,28.110,154.805
C00803=1081.381,369.383,402.061,176.377,28.104,154.804
C00804=1081.375,369.135,402.099,176.373,28.097,154.803
C00805=1081.368,368.888,402.135,176.370,28.092,154.802
C00806=1081.363,368.641,402.172,176.366,28.085,154.801
C00807=1081.357,368.394,402.209,176.363,28.079,154.799
C00808=1081.350,368.147,402.246,176.360,28.073,154.798
C00809=1081.344,367.900,402.283,176.356,28.067,154.797
C00810=1081.338,367.653,402.319,176.353,28.061,154.796
C00811=1081.332,367.406,402.356,176.349,28.054,154.795
C00812=1081.325,367.158,402.393,176.346,28.049,154.794
C00813=1081.319,366.911,402.430,176.342,28.042,154.793
C00814=1081.314,366.663,402.467,176.339,28.037,154.792
C00815=1081.307,366.416,402.503,176.335,28.030,154.791
C00816=1081.301,366.169,402.540,176.333,28.024,154.789
C00817=1081.295,365.922,402.577,176.329,28.018,154.788
C00818=1081.289,365.675,402.613,176.326,28.012,154.787
C00819=1081.283,365.428,402.650,176.323,28.007,154.786
C00820=1081.277,365.181,402.687,176.319,28.000,154.785
C00821=1081.271,364.933,402.723,176.316,27.994,154.784
C00822=1081.264,364.686,402.759,176.312,27.989,154.783
C00823=1081.258,364.439,402.796,176.309,27.982,154.782
C00824=1081.252,364.192,402.832,176.305,27.976,154.781
C00825=1081.246,363.944,402.869,176.302,27.971,154.780
C00826=1081.240,363.697,402.905,176.299,27.965,154.779
C00827=1081.234,363.450,402.942,176.295,27.959,154.778
C00828=1081.227,363.203,402.978,176.292,27.953,154.776
C00829=1081.221,362.956,403.014,176.288,27.947,154.775
C00830=1081.215,362.708,403.050,176.285,27.941,154.774
C00831=1081.209,362.461,403.087,176.281,27.936,154.773
C00832=1081.202,362.214,403.123,176.278,27.930,154.772
C00833=1081.196,361.967,403.159,176.275,27.924,154.771
C00834=1081.190,361.720,403.195,176.271,27.918,154.770
C00835=1081.184,361.472,403.232,176.268,27.913,154.769
C00836=1081.178,361.225,403.268,176.265,27.907,154.768
C00837=1081.172,360.978,403.304,176.261,27.901,154.767
C00838=1081.166,360.730,403.340,176.258,27.895,154.766
C00839=1081.160,360.483,403.377,176.254,27.889,154.765
C00840=1081.154,360.235,403.412,176.251,27.884,154.764
C00841=1081.147,359.988,403.449,176.248,27.878,154.763
C00842=1081.141,359.740,403.485,176.244,27.872,154.762
C00843=1081.135,359.494,403.521,176.241,27.866,154.761
C00844=1081.129,359.246,403.556,176.239,27.861,154.760
C00845=1081.123,358.999,403.593,176.234,27.855,154.759
C00846=1081.117,358.752,403.629,176.232,27.850,154.758
C00847=1081.110,358.505,403.664,176.228,27.844,154.757
C00848=1081.100,358.091,403.724,176.222,27.835,154.755
C00849=1081.090,357.678,403.784,176.217,27.825,154.754
C00850=1081.079,357.265,403.844,176.212,27.816,154.752
C00851=1081.069,356.851,403.903,176.206,27.807,154.750
C00852=1081.063,356.604,403.940,176.202,27.801,154.749
C00853=1081.057,356.357,403.975,176.199,27.795,154.748
C00854=1081.051,356.110,404.011,176.196,27.790,154.748
C00855=1081.045,355.862,404.047,176.192,27.784,154.747
C00856=1081.038,355.615,404.082,176.189,27.779,154.746
C00857=1081.033,355.368,404.118,176.186,27.773,154.745
C00858=1081.027,355.121,404.154,176.182,27.768,154.744
C00859=1081.021,354.873,404.189,176.179,27.762,154.743
C00860=1081.015,354.625,404.225,176.176,27.757,154.742
C00861=1081.008,354.378,404.260,176.172,27.751,154.741
C00862=1081.002,354.131,404.296,176.169,27.746,154.740
C00863=1080.996,353.883,404.331,176.166,27.740,154.739
C00864=1080.990,353.636,404.367,176.163,27.735,154.738
C00865=1080.984,353.389,404.402,176.159,27.730,154.737
C00866=1080.978,353.141,404.438,176.156,27.724,154.736
C00867=1080.972,352.894,404.473,176.153,27.719,154.735
C00868=1080.966,352.646,404.509,176.149,27.713,154.734
C00869=1080.960,352.399,404.544,176.146,27.708,154.733
C00870=1080.954,352.152,404.579,176.143,27.702,154.732
C00871=1080.947,351.904,404.615,176.140,27.697,154.731
C00872=1080.942,351.657,404.650,176.136,27.692,154.730
C00873=1080.936,351.409,404.685,176.133,27.686,154.729
C00874=1080.929,351.162,404.720,176.130,27.681,154.729
C00875=1080.923,350.914,404.756,176.127,27.676,154.728
C00876=1080.917,350.667,404.791,176.123,27.671,154.727
C00877=1080.911,350.420,404.826,176.120,27.665,154.726
C00878=1080.905,350.172,404.861,176.117,27.660,154.725
C00879=1080.899,349.925,404.896,176.114,27.654,154.724
C00880=1080.893,349.677,404.932,176.110,27.649,154.723
C00881=1080.887,349.430,404.967,176.107,27.644,154.722
C00882=1080.881,349.182,405.002,176.104,27.639,154.721
C00883=1080.874,348.935,405.037,176.101,27.633,154.720
C00884=1080.869,348.688,405.072,176.097,27.628,154.719
C00885=1080.863,348.440,405.107,176.094,27.623,154.718
C00886=1080.857,348.193,405.142,176.091,27.618,154.718
C00887=1080.851,347.945,405.176,176.088,27.613,154.717
C00888=1080.845,347.697,405.212,176.085,27.608,154.716
C00889=1080.839,347.450,405.246,176.081,27.602,154.715
C00890=1080.832,347.202,405.281,176.078,27.597,154.714
C00891=1080.827,346.955,405.316,176.075,27.592,154.713
C00892=1080.820,346.707,405.351,176.072,27.586,154.712
C00893=1080.815,346.460,405.386,176.069,27.582,154.711
C00894=1080.808,346.212,405.421,176.065,27.576,154.711
C00895=1080.803,345.965,405.455,176.062,27.571,154.710
C00896=1080.796,345.717,405.491,176.059,27.566,154.709
C00897=1080.790,345.469,405.525,176.056,27.561,154.708
C00898=1080.784,345.223,405.560,176.053,27.556,154.707
C00899=1080.778,344.975,405.595,176.050,27.551,154.706
C00900=1080.768,344.565,405.652,176.044,27.542,154.705
C00901=1080.759,344.155,405.710,176.039,27.534,154.703
C00902=1080.749,343.744,405.767,176.034,27.525,154.702
C00903=1080.739,343.334,405.824,176.028,27.517,154.701
C00904=1080.732,343.086,405.858,176.025,27.512,154.700
C00905=1080.726,342.839,405.892,176.022,27.507,154.699
C00906=1080.719,342.592,405.928,176.018,27.502,154.698
C00907=1080.714,342.344,405.962,176.015,27.497,154.697
C00908=1080.708,342.096,405.997,176.012,27.492,154.696
C00909=1080.702,341.849,406.031,176.009,27.487,154.696
C00910=1080.696,341.602,406.065,176.006,27.482,154.695
C00911=1080.690,341.354,406.099,176.003,27.477,154.694
C00912=1080.685,341.106,406.134,176.000,27.472,154.693
C00913=1080.678,340.859,406.169,175.996,27.467,154.692
C00914=1080.672,340.611,406.203,175.993,27.462,154.691
C00915=1080.666,340.364,406.237,175.990,27.457,154.691
C00916=1080.660,340.116,406.272,175.986,27.452,154.690
C00917=1080.654,339.869,406.306,175.983,27.447,154.689
C00918=1080.647,339.621,406.340,175.980,27.442,154.688
C00919=1080.642,339.373,406.375,175.977,27.437,154.687
C00920=1080.636,339.126,406.409,175.974,27.432,154.686
C00921=1080.630,338.877,406.442,175.971,27.427,154.686
C00922=1080.624,338.630,406.476,175.967,27.422,154.685
C00923=1080.618,338.383,406.510,175.964,27.417,154.684
C00924=1080.612,338.135,406.545,175.961,27.412,154.683
C00925=1080.606,337.888,406.579,175.958,27.408,154.682
C00926=1080.600,337.640,406.613,175.955,27.403,154.682
C00927=1080.594,337.392,406.647,175.952,27.398,154.681
C00928=1080.588,337.144,406.681,175.949,27.393,154.680
C00929=1080.582,336.897,406.715,175.946,27.388,154.679
C00930=1080.576,336.649,406.749,175.943,27.383,154.678
C00931=1080.570,336.402,406.783,175.940,27.379,154.678
C00932=1080.564,336.154,406.817,175.937,27.374,154.677
C00933=1080.559,335.907,406.851,175.933,27.369,154.676
C00934=1080.552,335.659,406.885,175.929,27.364,154.675
C00935=1080.546,335.412,406.919,175.926,27.359,154.674
C00936=1080.540,335.164,406.952,175.923,27.355,154.674
C00937=1080.534,334.916,406.986,175.920,27.350,154.673
C00938=1080.528,334.668,407.020,175.917,27.345,154.672
C00939=1080.522,334.421,407.054,175.914,27.340,154.671
C00940=1080.516,334.173,407.088,175.911,27.336,154.671
C00941=1080.511,333.925,407.121,175.908,27.331,154.670
C00942=1080.504,333.677,407.156,175.905,27.326,154.669
C00943=1080.498,333.430,407.188,175.902,27.321,154.668
C00944=1080.492,333.183,407.222,175.899,27.317,154.667
C00945=1080.487,332.935,407.256,175.896,27.312,154.667
C00946=1080.481,332.687,407.290,175.893,27.307,154.666
C00947=1080.475,332.439,407.323,175.890,27.302,154.665
C00948=1080.469,332.192,407.357,175.886,27.298,154.664
C00949=1080.463,331.944,407.391,175.883,27.293,154.664
C00950=1080.456,331.697,407.424,175.880,27.288,154.663
C00951=1080.451,331.449,407.458,175.877,27.283,154.662
C00952=1080.440,331.033,407.514,175.872,27.276,154.661
C00953=1080.430,330.618,407.570,175.866,27.268,154.660
C00954=1080.420,330.202,407.626,175.862,27.261,154.658
C00955=1080.410,329.786,407.682,175.856,27.253,154.657
C00956=1080.404,329.539,407.715,175.853,27.248,154.656
C00957=1080.397,329.290,407.748,175.850,27.243,154.656
C00958=1080.391,329.043,407.782,175.847,27.239,154.655
C00959=1080.385,328.795,407.815,175.844,27.234,154.654
C00960=1080.379,328.548,407.848,175.841,27.230,154.653
C00961=1080.373,328.300,407.881,175.838,27.225,154.653
C00962=1080.367,328.052,407.914,175.835,27.221,154.652
C00963=1080.361,327.805,407.948,175.832,27.216,154.651
C00964=1080.354,327.557,407.981,175.828,27.212,154.651
C00965=1080.349,327.309,408.014,175.825,27.207,154.650
C00966=1080.343,327.061,408.047,175.822,27.203,154.649
C00967=1080.337,326.813,408.081,175.819,27.198,154.648
C00968=1080.331,326.566,408.113,175.816,27.194,154.648
C00969=1080.325,326.318,408.147,175.813,27.189,154.647
C00970=1080.319,326.070,408.179,175.810,27.185,154.646
C00971=1080.313,325.822,408.213,175.807,27.180,154.645
C00972=1080.307,325.575,408.245,175.804,27.175,154.645
C00973=1080.301,325.327,408.278,175.801,27.171,154.644
C00974=1080.295,325.079,408.312,175.797,27.166,154.643
C00975=1080.289,324.832,408.344,175.794,27.162,154.643
C00976=1080.283,324.584,408.378,175.792,27.158,154.642
C00977=1080.277,324.336,408.410,175.789,27.153,154.641
C00978=1080.271,324.088,408.444,175.786,27.149,154.641
C00979=1080.265,323.841,408.476,175.783,27.144,154.640
C00980=1080.259,323.593,408.509,175.780,27.140,154.639
C00981=1080.253,323.345,408.543,175.777,27.135,154.638
C00982=1080.247,323.097,408.575,175.774,27.131,154.638
C00983=1080.242,322.849,408.608,175.771,27.126,154.637
C00984=1080.236,322.601,408.641,175.767,27.122,154.636
C00985=1080.229,322.354,408.673,175.764,27.117,154.636
C00986=1080.224,322.106,408.707,175.761,27.113,154.635
C00987=1080.218,321.858,408.739,175.758,27.108,154.634
C00988=1080.212,321.611,408.771,175.755,27.104,154.634
C00989=1080.206,321.363,408.804,175.753,27.100,154.633
C00990=1080.200,321.115,408.837,175.750,27.095,154.632
C00991=1080.194,320.867,408.869,175.747,27.091,154.631
C00992=1080.189,320.619,408.903,175.744,27.086,154.631
C00993=1080.182,320.372,408.935,175.740,27.082,154.630
C00994=1080.176,320.123,408.967,175.737,27.077,154.629
C00995=1080.171,319.876,409.000,175.734,27.073,154.629
C00996=1080.165,319.629,409.033,175.731,27.068,154.628
C00997=1080.159,319.380,409.065,175.728,27.064,154.627
C00998=1080.154,319.132,409.098,175.725,27.059,154.627
C00999=1080.148,318.884,409.130,175.723,27.055,154.626
C01000=1080.142,318.637,409.163,175.720,27.051,154.625
C01001=1080.137,318.389,409.195,175.717,27.046,154.624
C01002=1080.130,318.141,409.228,175.714,27.042,154.624
C01003=1080.124,317.894,409.261,175.710,27.038,154.623
C01004=1080.120,317.682,409.288,175.708,27.034,154.622
C01005=1080.115,317.471,409.316,175.706,27.030,154.622
C01006=1080.109,317.260,409.343,175.703,27.026,154.621
C01007=1080.105,317.049,409.371,175.701,27.022,154.621
C01008=1080.100,316.839,409.399,175.698,27.019,154.620
C01009=1080.095,316.626,409.426,175.695,27.015,154.620
C01010=1080.090,316.416,409.454,175.693,27.011,154.619
C01011=1080.086,316.205,409.482,175.691,27.008,154.618
C01012=1080.080,315.957,409.514,175.687,27.003,154.618
C01013=1080.073,315.709,409.546,175.684,26.999,154.617
C01014=1080.068,315.461,409.578,175.681,26.994,154.616
C01015=1080.062,315.214,409.611,175.678,26.990,154.616
C01016=1080.056,314.965,409.643,175.676,26.986,154.615
C01017=1080.051,314.718,409.675,175.673,26.982,154.614
C01018=1080.045,314.470,409.707,175.670,26.977,154.614
C01019=1080.039,314.222,409.740,175.667,26.973,154.613
C01020=1080.032,313.974,409.771,175.663,26.969,154.612
C01021=1080.026,313.726,409.803,175.660,26.965,154.612
C01022=1080.021,313.478,409.835,175.658,26.961,154.611
C01023=1080.014,313.231,409.868,175.655,26.956,154.610
C01024=1080.008,312.983,409.900,175.652,26.952,154.610
C01025=1080.002,312.734,409.932,175.649,26.948,154.609
C01026=1079.996,312.487,409.963,175.646,26.944,154.609
C01027=1079.990,312.239,409.995,175.643,26.940,154.608
C01028=1079.984,311.991,410.027,175.640,26.936,154.607
C01029=1079.979,311.743,410.059,175.637,26.931,154.607
C01030=1079.972,311.496,410.091,175.634,26.927,154.606
C01031=1079.966,311.248,410.123,175.631,26.923,154.605
C01032=1079.960,311.000,410.154,175.628,26.919,154.605
C01033=1079.954,310.752,410.186,175.625,26.915,154.604
C01034=1079.948,310.504,410.218,175.622,26.911,154.604
C01035=1079.942,310.257,410.249,175.619,26.906,154.603
C01036=1079.936,310.008,410.281,175.616,26.902,154.602
C01037=1079.930,309.760,410.314,175.613,26.898,154.602
C01038=1079.925,309.513,410.345,175.610,26.894,154.601
C01039=1079.918,309.265,410.377,175.608,26.890,154.600
C01040=1079.913,309.017,410.408,175.605,26.886,154.600
C01041=1079.907,308.769,410.440,175.602,26.881,154.599
C01042=1079.900,308.521,410.472,175.598,26.877,154.599
C01043=1079.895,308.274,410.503,175.595,26.873,154.598
C01044=1079.889,308.025,410.535,175.593,26.869,154.597
C01045=1079.884,307.777,410.566,175.590,26.865,154.597
C01046=1079.877,307.529,410.598,175.587,26.860,154.596
C01047=1079.872,307.282,410.629,175.584,26.856,154.595
C01048=1079.866,307.034,410.661,175.581,26.852,154.595
C01049=1079.859,306.786,410.693,175.578,26.848,154.594
C01050=1079.854,306.538,410.724,175.575,26.844,154.594
C01051=1079.848,306.290,410.756,175.572,26.840,154.593
C01052=1079.842,306.042,410.787,175.569,26.836,154.592
C01053=1079.836,305.795,410.819,175.567,26.832,154.592
C01054=1079.830,305.546,410.851,175.564,26.828,154.591
C01055=1079.824,305.299,410.881,175.561,26.823,154.590
C01056=1079.818,305.050,410.913,175.557,26.819,154.590
C01057=1079.813,304.803,410.945,175.554,26.815,154.589
C01058=1079.807,304.554,410.975,175.552,26.811,154.589
C01059=1079.801,304.307,411.007,175.549,26.807,154.588
C01060=1079.791,303.888,411.060,175.544,26.800,154.587
C01061=1079.782,303.469,411.113,175.539,26.793,154.586
C01062=1079.771,303.050,411.166,175.534,26.786,154.585
C01063=1079.762,302.631,411.219,175.530,26.780,154.584
C01064=1079.756,302.382,411.250,175.527,26.775,154.583
C01065=1079.750,302.135,411.281,175.524,26.771,154.583
C01066=1079.744,301.886,411.312,175.521,26.767,154.582
C01067=1079.738,301.639,411.344,175.518,26.763,154.581
C01068=1079.733,301.391,411.374,175.515,26.759,154.581
C01069=1079.727,301.143,411.406,175.512,26.754,154.580
C01070=1079.721,300.895,411.437,175.509,26.751,154.580
C01071=1079.716,300.647,411.469,175.507,26.747,154.579
C01072=1079.710,300.399,411.499,175.504,26.742,154.578
C01073=1079.705,300.151,411.530,175.501,26.738,154.578
C01074=1079.698,299.903,411.561,175.497,26.734,154.577
C01075=1079.693,299.655,411.592,175.495,26.730,154.577
C01076=1079.687,299.407,411.623,175.492,26.726,154.576
C01077=1079.682,299.159,411.655,175.489,26.722,154.575
C01078=1079.676,298.911,411.685,175.487,26.718,154.575
C01079=1079.670,298.664,411.717,175.484,26.713,154.574
C01080=1079.664,298.415,411.747,175.481,26.710,154.574
C01081=1079.659,298.167,411.778,175.478,26.706,154.573
C01082=1079.653,297.919,411.809,175.475,26.701,154.572
C01083=1079.648,297.672,411.840,175.472,26.697,154.572
C01084=1079.641,297.423,411.871,175.469,26.693,154.571
C01085=1079.635,297.176,411.901,175.467,26.690,154.571
C01086=1079.630,296.927,411.932,175.464,26.685,154.570
C01087=1079.624,296.679,411.963,175.461,26.681,154.569
C01088=1079.618,296.432,411.994,175.458,26.677,154.569
C01089=1079.612,296.184,412.024,175.455,26.674,154.568
C01090=1079.606,295.935,412.056,175.452,26.670,154.568
C01091=1079.600,295.687,412.086,175.450,26.666,154.567
C01092=1079.595,295.439,412.116,175.447,26.662,154.566
C01093=1079.589,295.192,412.147,175.444,26.658,154.566
C01094=1079.583,294.943,412.178,175.441,26.654,154.565
C01095=1079.577,294.695,412.208,175.438,26.650,154.565
C01096=1079.572,294.447,412.239,175.435,26.646,154.564
C01097=1079.566,294.199,412.269,175.433,26.642,154.564
C01098=1079.559,293.951,412.300,175.430,26.638,154.563
C01099=1079.553,293.703,412.330,175.427,26.634,154.562
C01100=1079.548,293.455,412.361,175.425,26.630,154.562
C01101=1079.543,293.207,412.392,175.421,26.626,154.561
C01102=1079.537,292.959,412.422,175.418,26.622,154.561
C01103=1079.530,292.711,412.453,175.416,26.618,154.560
C01104=1079.525,292.463,412.483,175.413,26.615,154.560
C01105=1079.519,292.215,412.513,175.410,26.610,154.559
C01106=1079.513,291.967,412.544,175.408,26.607,154.558
C01107=1079.507,291.719,412.574,175.404,26.603,154.558
C01108=1079.501,291.471,412.605,175.401,26.598,154.557
C01109=1079.496,291.223,412.636,175.399,26.595,154.557
C01110=1079.490,290.974,412.665,175.396,26.591,154.556
C01111=1079.484,290.726,412.696,175.393,26.587,154.556
C01112=1079.474,290.322,412.745,175.388,26.581,154.555
C01113=1079.465,289.917,412.795,175.385,26.574,154.554
C01114=1079.455,289.512,412.844,175.380,26.568,154.553
C01115=1079.446,289.108,412.893,175.375,26.561,154.552
C01116=1079.440,288.859,412.923,175.372,26.558,154.551
C01117=1079.434,288.612,412.954,175.369,26.554,154.551
C01118=1079.428,288.363,412.983,175.367,26.550,154.550
C01119=1079.423,288.115,413.014,175.364,26.546,154.550
C01120=1079.417,287.868,413.044,175.361,26.542,154.549
C01121=1079.411,287.619,413.074,175.358,26.538,154.549
C01122=1079.405,287.372,413.103,175.355,26.535,154.548
C01123=1079.399,287.123,413.133,175.353,26.531,154.548
C01124=1079.393,286.875,413.164,175.350,26.527,154.547
C01125=1079.387,286.627,413.194,175.347,26.523,154.546
C01126=1079.381,286.378,413.224,175.344,26.519,154.546
C01127=1079.376,286.131,413.254,175.341,26.515,154.545
C01128=1079.370,285.882,413.284,175.339,26.512,154.545
C01129=1079.364,285.635,413.313,175.336,26.508,154.544
C01130=1079.358,285.386,413.343,175.333,26.504,154.544
C01131=1079.352,285.138,413.373,175.331,26.500,154.543
C01132=1079.347,284.890,413.403,175.327,26.496,154.543
C01133=1079.341,284.642,413.433,175.325,26.492,154.542
C01134=1079.335,284.394,413.462,175.322,26.488,154.541
C01135=1079.329,284.146,413.493,175.320,26.485,154.541
C01136=1079.323,283.898,413.522,175.317,26.481,154.540
C01137=1079.318,283.649,413.552,175.314,26.477,154.540
C01138=1079.312,283.401,413.582,175.312,26.473,154.539
C01139=1079.306,283.153,413.611,175.308,26.469,154.539
C01140=1079.300,282.905,413.641,175.306,26.466,154.538
C01141=1079.294,282.657,413.671,175.303,26.462,154.538
C01142=1079.289,282.409,413.701,175.300,26.457,154.537
C01143=1079.283,282.160,413.731,175.298,26.454,154.536
C01144=1079.277,281.913,413.760,175.295,26.450,154.536
C01145=1079.271,281.664,413.790,175.292,26.446,154.535
C01146=1079.266,281.416,413.820,175.289,26.443,154.535
C01147=1079.260,281.168,413.850,175.287,26.439,154.534
C01148=1079.254,280.920,413.879,175.284,26.435,154.534
C01149=1079.249,280.672,413.908,175.282,26.431,154.533
C01150=1079.243,280.424,413.938,175.279,26.427,154.533
C01151=1079.237,280.175,413.967,175.275,26.423,154.532
C01152=1079.232,279.927,413.997,175.273,26.420,154.532
C01153=1079.225,279.680,414.026,175.270,26.416,154.531
C01154=1079.219,279.431,414.056,175.268,26.412,154.531
C01155=1079.213,279.183,414.085,175.265,26.409,154.530
C01156=1079.208,278.935,414.115,175.263,26.405,154.529
C01157=1079.202,278.686,414.144,175.259,26.401,154.529
C01158=1079.196,278.438,414.173,175.257,26.397,154.528
C01159=1079.190,278.189,414.203,175.254,26.393,154.528
C01160=1079.184,277.941,414.232,175.251,26.389,154.527
C01161=1079.179,277.693,414.262,175.249,26.386,154.527
C01162=1079.173,277.445,414.290,175.246,26.382,154.526
C01163=1079.168,277.197,414.320,175.243,26.378,154.526
C01164=1079.158,276.802,414.367,175.239,26.372,154.525
C01165=1079.149,276.407,414.414,175.235,26.367,154.524
C01166=1079.140,276.012,414.460,175.230,26.360,154.523
C01167=1079.130,275.618,414.507,175.226,26.354,154.522
C01168=1079.125,275.369,414.536,175.224,26.350,154.522
C01169=1079.118,275.121,414.565,175.220,26.346,154.521
C01170=1079.114,274.873,414.594,175.218,26.343,154.521
C01171=1079.107,274.625,414.623,175.215,26.339,154.520
C01172=1079.101,274.376,414.652,175.213,26.335,154.520
C01173=1079.096,274.128,414.682,175.210,26.332,154.519
C01174=1079.089,273.880,414.711,175.207,26.328,154.519
C01175=1079.085,273.632,414.740,175.204,26.324,154.518
C01176=1079.079,273.383,414.768,175.202,26.321,154.518
C01177=1079.072,273.135,414.797,175.199,26.317,154.517
C01178=1079.067,272.887,414.827,175.197,26.313,154.517
C01179=1079.061,272.639,414.856,175.194,26.309,154.516
C01180=1079.055,272.391,414.884,175.191,26.306,154.516
C01181=1079.050,272.142,414.914,175.188,26.302,154.515
C01182=1079.043,271.894,414.943,175.186,26.298,154.514
C01183=1079.038,271.645,414.971,175.183,26.294,154.514
C01184=1079.033,271.398,415.000,175.181,26.291,154.513
C01185=1079.026,271.149,415.029,175.178,26.287,154.513
C01186=1079.020,270.901,415.058,175.175,26.283,154.512
C01187=1079.014,270.653,415.087,175.172,26.279,154.512
C01188=1079.009,270.405,415.116,175.170,26.276,154.511
C01189=1079.003,270.156,415.144,175.167,26.272,154.511
C01190=1078.997,269.908,415.173,175.165,26.268,154.510
C01191=1078.991,269.659,415.202,175.162,26.265,154.510
C01192=1078.986,269.411,415.231,175.159,26.261,154.509
C01193=1078.980,269.163,415.260,175.156,26.257,154.509
C01194=1078.974,268.915,415.288,175.154,26.254,154.508
C01195=1078.968,268.667,415.317,175.151,26.250,154.508
C01196=1078.962,268.418,415.345,175.149,26.246,154.507
C01197=1078.957,268.170,415.375,175.147,26.243,154.507
C01198=1078.951,267.921,415.403,175.143,26.239,154.506
C01199=1078.945,267.674,415.432,175.141,26.236,154.506
C01200=1078.939,267.425,415.460,175.138,26.232,154.505
C01201=1078.933,267.176,415.488,175.136,26.228,154.505
C01202=1078.928,266.929,415.517,175.133,26.224,154.504
C01203=1078.922,266.680,415.545,175.130,26.221,154.504
C01204=1078.916,266.432,415.575,175.127,26.217,154.503
C01205=1078.911,266.184,415.603,175.125,26.213,154.503
C01206=1078.905,265.935,415.631,175.122,26.209,154.502
C01207=1078.899,265.687,415.660,175.120,26.206,154.502
C01208=1078.893,265.439,415.688,175.117,26.202,154.501
C01209=1078.888,265.190,415.717,175.114,26.198,154.501
C01210=1078.882,264.942,415.745,175.112,26.195,154.500
C01211=1078.876,264.694,415.774,175.109,26.191,154.499
C01212=1078.870,264.445,415.802,175.107,26.187,154.499
C01213=1078.864,264.198,415.831,175.104,26.183,154.498
C01214=1078.858,263.949,415.859,175.102,26.180,154.498
C01215=1078.853,263.701,415.887,175.098,26.176,154.498
C01216=1078.843,263.309,415.932,175.095,26.171,154.497
C01217=1078.834,262.917,415.977,175.091,26.165,154.496
C01218=1078.825,262.525,416.021,175.086,26.159,154.495
C01219=1078.815,262.133,416.065,175.083,26.154,154.494
C01220=1078.810,261.885,416.094,175.079,26.150,154.494
C01221=1078.804,261.636,416.122,175.077,26.146,154.493
C01222=1078.798,261.388,416.150,175.074,26.143,154.493
C01223=1078.792,261.140,416.178,175.072,26.139,154.492
C01224=1078.786,260.891,416.206,175.070,26.136,154.492
C01225=1078.780,260.643,416.234,175.066,26.132,154.491
C01226=1078.774,260.394,416.262,175.064,26.128,154.491
C01227=1078.768,260.146,416.291,175.061,26.124,154.490
C01228=1078.762,259.898,416.318,175.059,26.121,154.490
C01229=1078.756,259.649,416.346,175.056,26.117,154.489
C01230=1078.751,259.401,416.374,175.054,26.114,154.489
C01231=1078.745,259.152,416.403,175.051,26.110,154.488
C01232=1078.739,258.905,416.430,175.048,26.106,154.488
C01233=1078.733,258.656,416.458,175.046,26.103,154.487
C01234=1078.728,258.408,416.486,175.043,26.099,154.487
C01235=1078.722,258.159,416.515,175.041,26.096,154.486
C01236=1078.716,257.911,416.542,175.039,26.092,154.486
C01237=1078.710,257.663,416.570,175.035,26.088,154.485
C01238=1078.705,257.414,416.597,175.033,26.085,154.485
C01239=1078.698,257.165,416.625,175.030,26.081,154.485
C01240=1078.693,256.917,416.653,175.028,26.078,154.484
C01241=1078.687,256.669,416.681,175.026,26.074,154.483
C01242=1078.681,256.421,416.709,175.023,26.070,154.483
C01243=1078.675,256.172,416.737,175.020,26.067,154.482
C01244=1078.670,255.924,416.764,175.018,26.063,154.482
C01245=1078.664,255.675,416.793,175.015,26.060,154.482
C01246=1078.658,255.427,416.820,175.013,26.056,154.481
C01247=1078.652,255.179,416.848,175.010,26.052,154.480
C01248=1078.646,254.930,416.876,175.007,26.049,154.480
C01249=1078.641,254.682,416.903,175.005,26.045,154.479
C01250=1078.635,254.433,416.931,175.002,26.041,154.479
C01251=1078.629,254.185,416.959,175.000,26.038,154.479
C01252=1078.624,253.937,416.986,174.998,26.034,154.478
C01253=1078.618,253.688,417.014,174.995,26.030,154.477
C01254=1078.612,253.440,417.042,174.992,26.027,154.477
C01255=1078.606,253.191,417.069,174.989,26.023,154.476
C01256=1078.601,252.943,417.097,174.987,26.019,154.476
C01257=1078.595,252.695,417.125,174.985,26.016,154.475
C01258=1078.589,252.446,417.152,174.982,26.012,154.475
C01259=1078.584,252.198,417.180,174.980,26.009,154.474
C01260=1078.578,251.949,417.207,174.977,26.005,154.474
C01261=1078.572,251.701,417.235,174.974,26.001,154.473
C01262=1078.567,251.452,417.263,174.972,25.998,154.473
C01263=1078.561,251.204,417.290,174.970,25.994,154.472
C01264=1078.555,250.955,417.318,174.967,25.990,154.472
C01265=1078.550,250.707,417.345,174.965,25.987,154.471
C01266=1078.544,250.459,417.373,174.962,25.983,154.471
C01267=1078.538,250.210,417.400,174.959,25.980,154.470
C01268=1078.529,249.815,417.444,174.956,25.974,154.470
C01269=1078.520,249.421,417.487,174.952,25.968,154.469
C01270=1078.511,249.026,417.530,174.948,25.962,154.468
C01271=1078.502,248.632,417.574,174.944,25.956,154.467
C01272=1078.497,248.384,417.602,174.942,25.953,154.467
C01273=1078.491,248.135,417.629,174.938,25.949,154.466
C01274=1078.485,247.887,417.657,174.936,25.945,154.466
C01275=1078.480,247.638,417.683,174.934,25.942,154.465
C01276=1078.474,247.390,417.711,174.931,25.938,154.465
C01277=1078.468,247.142,417.738,174.929,25.934,154.464
C01278=1078.463,246.892,417.766,174.927,25.931,154.464
C01279=1078.457,246.644,417.792,174.924,25.927,154.463
C01280=1078.452,246.396,417.820,174.921,25.924,154.463
C01281=1078.446,246.148,417.847,174.919,25.920,154.462
C01282=1078.440,245.899,417.874,174.916,25.916,154.462
C01283=1078.434,245.650,417.901,174.914,25.912,154.461
C01284=1078.428,245.402,417.928,174.912,25.909,154.461
C01285=1078.423,245.154,417.955,174.910,25.906,154.460
C01286=1078.418,244.905,417.982,174.906,25.902,154.460
C01287=1078.411,244.656,418.009,174.904,25.898,154.459
C01288=1078.405,244.408,418.036,174.902,25.895,154.459
C01289=1078.400,244.160,418.064,174.899,25.891,154.458
C01290=1078.394,243.911,418.091,174.897,25.887,154.458
C01291=1078.389,243.663,418.117,174.895,25.884,154.457
C01292=1078.383,243.414,418.145,174.892,25.880,154.457
C01293=1078.377,243.165,418.171,174.889,25.876,154.456
C01294=1078.371,242.917,418.198,174.887,25.873,154.456
C01295=1078.366,242.669,418.225,174.885,25.870,154.455
C01296=1078.361,242.420,418.252,174.882,25.866,154.455
C01297=1078.355,242.171,418.279,174.880,25.862,154.454
C01298=1078.348,241.922,418.306,174.878,25.858,154.454
C01299=1078.343,241.674,418.332,174.874,25.855,154.453
C01300=1078.337,241.426,418.359,174.872,25.851,154.453
C01301=1078.331,241.177,418.386,174.870,25.848,154.452
C01302=1078.325,240.929,418.412,174.868,25.844,154.452
C01303=1078.320,240.680,418.439,174.865,25.841,154.451
C01304=1078.314,240.431,418.466,174.863,25.837,154.451
C01305=1078.308,240.183,418.493,174.860,25.834,154.450
C01306=1078.302,239.935,418.520,174.857,25.830,154.450
C01307=1078.297,239.686,418.546,174.855,25.826,154.449
C01308=1078.291,239.438,418.573,174.853,25.823,154.449
C01309=1078.285,239.189,418.600,174.851,25.819,154.448
C01310=1078.279,238.941,418.626,174.848,25.815,154.448
C01311=1078.273,238.692,418.653,174.845,25.812,154.447
C01312=1078.267,238.444,418.680,174.843,25.809,154.447
C01313=1078.262,238.195,418.706,174.841,25.805,154.446
C01314=1078.256,237.946,418.733,174.838,25.801,154.446
C01315=1078.250,237.698,418.759,174.836,25.798,154.445
C01316=1078.244,237.450,418.786,174.834,25.794,154.445
C01317=1078.239,237.201,418.813,174.831,25.791,154.444
C01318=1078.233,236.953,418.839,174.828,25.787,154.444
C01319=1078.227,236.704,418.865,174.826,25.784,154.444
C01320=1078.218,236.303,418.909,174.823,25.778,154.443
C01321=1078.209,235.901,418.952,174.819,25.772,154.442
C01322=1078.200,235.500,418.993,174.814,25.766,154.441
C01323=1078.191,235.099,419.037,174.811,25.760,154.440
C01324=1078.185,234.850,419.063,174.808,25.757,154.440
C01325=1078.180,234.602,419.089,174.806,25.753,154.439
C01326=1078.174,234.353,419.116,174.803,25.749,154.439
C01327=1078.168,234.104,419.142,174.801,25.745,154.438
C01328=1078.162,233.856,419.168,174.799,25.742,154.438
C01329=1078.156,233.608,419.195,174.797,25.739,154.437
C01330=1078.151,233.359,419.221,174.794,25.735,154.437
C01331=1078.145,233.111,419.247,174.792,25.731,154.436
C01332=1078.139,232.862,419.273,174.789,25.728,154.436
C01333=1078.134,232.613,419.300,174.787,25.724,154.435
C01334=1078.128,232.364,419.326,174.785,25.721,154.435
C01335=1078.122,232.116,419.352,174.782,25.717,154.434
C01336=1078.116,231.868,419.379,174.780,25.714,154.434
C01337=1078.110,231.619,419.404,174.778,25.710,154.433
C01338=1078.105,231.371,419.431,174.775,25.706,154.433
C01339=1078.099,231.122,419.457,174.772,25.702,154.432
C01340=1078.094,230.873,419.483,174.770,25.699,154.432
C01341=1078.088,230.624,419.510,174.768,25.696,154.431
C01342=1078.082,230.376,419.535,174.766,25.692,154.431
C01343=1078.076,230.127,419.562,174.764,25.688,154.430
C01344=1078.071,229.879,419.587,174.761,25.685,154.430
C01345=1078.065,229.631,419.614,174.758,25.681,154.430
C01346=1078.059,229.382,419.639,174.756,25.678,154.429
C01347=1078.054,229.133,419.665,174.754,25.674,154.428
C01348=1078.048,228.885,419.692,174.752,25.671,154.428
C01349=1078.042,228.636,419.717,174.749,25.667,154.428
C01350=1078.036,228.387,419.743,174.747,25.663,154.427
C01351=1078.030,228.139,419.770,174.745,25.660,154.427
C01352=1078.024,227.890,419.795,174.742,25.657,154.426
C01353=1078.019,227.641,419.821,174.740,25.653,154.426
C01354=1078.012,227.393,419.847,174.737,25.649,154.425
C01355=1078.007,227.144,419.873,174.735,25.645,154.425
C01356=1078.002,226.896,419.898,174.733,25.642,154.424
C01357=1077.996,226.647,419.924,174.731,25.639,154.424
C01358=1077.990,226.399,419.950,174.728,25.635,154.423
C01359=1077.985,226.150,419.976,174.725,25.631,154.423
C01360=1077.978,225.901,420.002,174.723,25.628,154.422
C01361=1077.973,225.652,420.028,174.721,25.624,154.422
C01362=1077.967,225.403,420.053,174.719,25.621,154.421
C01363=1077.961,225.156,420.079,174.717,25.617,154.421
C01364=1077.955,224.907,420.105,174.715,25.614,154.420
C01365=1077.950,224.658,420.131,174.712,25.610,154.420
C01366=1077.944,224.409,420.157,174.709,25.606,154.419
C01367=1077.938,224.160,420.182,174.707,25.603,154.419
C01368=1077.933,223.912,420.207,174.705,25.600,154.418
C01369=1077.927,223.663,420.233,174.703,25.596,154.418
C01370=1077.921,223.415,420.259,174.701,25.592,154.417
C01371=1077.916,223.166,420.285,174.698,25.588,154.417
C01372=1077.906,222.757,420.327,174.694,25.582,154.416
C01373=1077.897,222.347,420.370,174.691,25.576,154.415
C01374=1077.887,221.937,420.412,174.687,25.571,154.414
C01375=1077.879,221.528,420.454,174.683,25.565,154.414
C01376=1077.872,221.279,420.479,174.680,25.561,154.413
C01377=1077.867,221.030,420.504,174.678,25.558,154.413
C01378=1077.861,220.781,420.530,174.676,25.554,154.412
C01379=1077.855,220.533,420.555,174.674,25.551,154.412
C01380=1077.849,220.284,420.580,174.672,25.547,154.411
C01381=1077.844,220.035,420.606,174.670,25.543,154.411
C01382=1077.838,219.787,420.631,174.667,25.540,154.410
C01383=1077.832,219.539,420.656,174.664,25.536,154.410
C01384=1077.827,219.290,420.682,174.662,25.533,154.409
C01385=1077.820,219.041,420.707,174.660,25.529,154.409
C01386=1077.814,218.792,420.733,174.658,25.526,154.408
C01387=1077.810,218.543,420.758,174.656,25.522,154.408
C01388=1077.803,218.295,420.783,174.654,25.519,154.407
C01389=1077.797,218.046,420.808,174.651,25.515,154.407
C01390=1077.792,217.798,420.834,174.648,25.511,154.406
C01391=1077.786,217.549,420.859,174.646,25.508,154.406
C01392=1077.780,217.300,420.884,174.644,25.504,154.405
C01393=1077.775,217.052,420.909,174.642,25.501,154.405
C01394=1077.769,216.803,420.935,174.640,25.497,154.404
C01395=1077.763,216.554,420.960,174.638,25.494,154.404
C01396=1077.757,216.306,420.985,174.636,25.490,154.403
C01397=1077.752,216.057,421.010,174.633,25.486,154.403
C01398=1077.746,215.808,421.036,174.631,25.483,154.402
C01399=1077.740,215.560,421.061,174.628,25.479,154.402
C01400=1077.734,215.311,421.085,174.626,25.476,154.401
C01401=1077.729,215.062,421.111,174.624,25.472,154.401
C01402=1077.723,214.814,421.136,174.622,25.468,154.400
C01403=1077.717,214.564,421.161,174.620,25.465,154.400
C01404=1077.712,214.317,421.186,174.617,25.462,154.399
C01405=1077.706,214.068,421.212,174.615,25.458,154.399
C01406=1077.700,213.818,421.236,174.613,25.454,154.398
C01407=1077.695,213.570,421.261,174.611,25.451,154.398
C01408=1077.689,213.321,421.286,174.608,25.447,154.397
C01409=1077.684,213.073,421.311,174.606,25.443,154.397
C01410=1077.678,212.824,421.337,174.604,25.440,154.396
C01411=1077.672,212.575,421.361,174.602,25.436,154.396
C01412=1077.666,212.327,421.386,174.600,25.432,154.395
C01413=1077.661,212.077,421.411,174.598,25.429,154.395
C01414=1077.655,211.830,421.436,174.595,25.426,154.394
C01415=1077.649,211.580,421.461,174.593,25.422,154.394
C01416=1077.643,211.332,421.486,174.591,25.418,154.393
C01417=1077.637,211.083,421.510,174.589,25.415,154.393
C01418=1077.632,210.835,421.535,174.587,25.412,154.392
C01419=1077.626,210.586,421.560,174.584,25.408,154.392
C01420=1077.620,210.336,421.584,174.582,25.404,154.391
C01421=1077.615,210.088,421.610,174.580,25.400,154.391
C01422=1077.609,209.839,421.635,174.577,25.397,154.390
C01423=1077.604,209.591,421.660,174.575,25.393,154.390
C01424=1077.594,209.185,421.700,174.572,25.387,154.389
C01425=1077.585,208.780,421.740,174.568,25.381,154.388
C01426=1077.576,208.374,421.780,174.565,25.376,154.388
C01427=1077.566,207.969,421.821,174.561,25.370,154.387
C01428=1077.542,206.932,421.920,174.451,25.312,154.388
C01429=1077.537,206.683,421.944,174.449,25.309,154.387
C01430=1077.531,206.435,421.969,174.447,25.307,154.387
C01431=1077.526,206.186,421.993,174.444,25.304,154.387
C01432=1077.520,205.937,422.017,174.442,25.301,154.386
C01433=1077.514,205.689,422.041,174.440,25.298,154.386
C01434=1077.509,205.439,422.065,174.437,25.296,154.386
C01435=1077.503,205.191,422.088,174.435,25.293,154.386
C01436=1077.497,204.942,422.113,174.433,25.290,154.385
C01437=1077.492,204.693,422.137,174.430,25.288,154.385
C01438=1077.486,204.445,422.161,174.428,25.285,154.385
C01439=1077.481,204.196,422.185,174.426,25.283,154.384
C01440=1077.476,203.947,422.209,174.423,25.280,154.384
C01441=1077.469,203.698,422.233,174.421,25.277,154.384
C01442=1077.464,203.449,422.256,174.419,25.275,154.384
C01443=1077.459,203.200,422.281,174.416,25.272,154.383
C01444=1077.453,202.952,422.304,174.414,25.269,154.383
C01445=1077.447,202.704,422.329,174.412,25.267,154.383
C01446=1077.442,202.454,422.352,174.409,25.264,154.383
C01447=1077.436,202.205,422.376,174.407,25.262,154.382
C01448=1077.430,201.956,422.399,174.404,25.259,154.382
C01449=1077.425,201.708,422.423,174.402,25.256,154.382
C01450=1077.418,201.459,422.447,174.401,25.255,154.382
C01451=1077.413,201.210,422.471,174.398,25.252,154.381
C01452=1077.407,200.961,422.495,174.396,25.249,154.381
C01453=1077.402,200.712,422.518,174.394,25.247,154.381
C01454=1077.396,200.464,422.542,174.391,25.244,154.381
C01455=1077.389,200.215,422.566,174.389,25.241,154.380
C01456=1077.384,199.966,422.589,174.386,25.239,154.380
C01457=1077.378,199.718,422.613,174.384,25.236,154.380
C01458=1077.373,199.468,422.637,174.382,25.234,154.379
C01459=1077.367,199.220,422.660,174.379,25.231,154.379
C01460=1077.362,198.971,422.683,174.377,25.229,154.379
C01461=1077.356,198.722,422.708,174.375,25.226,154.379
C01462=1077.350,198.473,422.731,174.372,25.224,154.379
C01463=1077.344,198.225,422.754,174.370,25.221,154.378
C01464=1077.339,197.975,422.778,174.368,25.219,154.378
C01465=1077.333,197.727,422.802,174.366,25.216,154.378
C01466=1077.328,197.478,422.825,174.364,25.213,154.377
C01467=1077.322,197.229,422.848,174.361,25.211,154.377
C01468=1077.316,196.980,422.872,174.359,25.208,154.377
C01469=1077.311,196.731,422.896,174.357,25.206,154.377
C01470=1077.305,196.483,422.919,174.354,25.203,154.376
C01471=1077.299,196.234,422.942,174.352,25.200,154.376
C01472=1077.294,195.984,422.966,174.349,25.198,154.376
C01473=1077.288,195.736,422.989,174.347,25.196,154.376
C01474=1077.282,195.487,423.012,174.346,25.193,154.375
C01475=1077.277,195.238,423.036,174.343,25.191,154.375
C01476=1077.271,194.990,423.060,174.341,25.188,154.375
C01477=1077.265,194.741,423.083,174.339,25.185,154.375
C01478=1077.260,194.492,423.106,174.336,25.183,154.374
C01479=1077.254,194.243,423.130,174.334,25.180,154.374
C01480=1077.249,193.995,423.153,174.332,25.177,154.374
C01481=1077.244,193.745,423.176,174.329,25.175,154.374
C01482=1077.237,193.497,423.200,174.328,25.173,154.373
C01483=1077.232,193.248,423.223,174.325,25.170,154.373
C01484=1077.226,192.999,423.246,174.323,25.167,154.373
C01485=1077.221,192.750,423.269,174.321,25.165,154.372
C01486=1077.215,192.502,423.293,174.318,25.162,154.372
C01487=1077.209,192.253,423.316,174.316,25.159,154.372
C01488=1077.204,192.004,423.339,174.314,25.157,154.372
C01489=1077.198,191.724,423.366,174.311,25.154,154.371
C01490=1077.192,191.443,423.392,174.309,25.151,154.371
C01491=1077.185,191.162,423.418,174.307,25.148,154.371
C01492=1077.179,190.882,423.444,174.305,25.146,154.370
C01493=1077.173,190.633,423.467,174.302,25.143,154.370
C01494=1077.168,190.384,423.490,174.300,25.140,154.370
C01495=1077.162,190.135,423.513,174.297,25.138,154.370
C01496=1077.157,189.886,423.537,174.295,25.135,154.369
C01497=1077.151,189.637,423.560,174.293,25.132,154.369
C01498=1077.145,189.388,423.583,174.291,25.130,154.369
C01499=1077.140,189.139,423.606,174.289,25.128,154.369
C01500=1077.134,188.890,423.629,174.287,25.125,154.368
C01501=1077.129,188.641,423.652,174.284,25.122,154.368
C01502=1077.123,188.393,423.676,174.282,25.120,154.368
C01503=1077.117,188.144,423.699,174.280,25.117,154.368
C01504=1077.112,187.896,423.721,174.278,25.115,154.367
C01505=1077.107,187.647,423.745,174.276,25.112,154.367
C01506=1077.101,187.398,423.768,174.274,25.109,154.367
C01507=1077.096,187.149,423.791,174.271,25.107,154.366
C01508=1077.090,186.900,423.814,174.269,25.104,154.366
C01509=1077.084,186.651,423.837,174.267,25.102,154.366
C01510=1077.079,186.401,423.859,174.265,25.099,154.366
C01511=1077.074,186.153,423.882,174.263,25.097,154.365
C01512=1077.069,185.904,423.905,174.260,25.094,154.365
C01513=1077.063,185.655,423.928,174.258,25.091,154.365
C01514=1077.057,185.406,423.951,174.257,25.089,154.365
C01515=1077.052,185.157,423.974,174.254,25.086,154.364
C01516=1077.046,184.908,423.997,174.252,25.084,154.364
C01517=1077.041,184.659,424.020,174.249,25.082,154.364
C01518=1077.034,184.411,424.043,174.247,25.079,154.364
C01519=1077.029,184.163,424.065,174.246,25.077,154.363
C01520=1077.024,183.913,424.087,174.243,25.074,154.363
C01521=1077.018,183.664,424.110,174.241,25.072,154.363
C01522=1077.012,183.415,424.133,174.239,25.069,154.363
C01523=1077.006,183.167,424.156,174.236,25.067,154.362
C01524=1077.000,182.918,424.179,174.235,25.064,154.362
C01525=1076.995,182.668,424.201,174.232,25.062,154.362
C01526=1076.989,182.419,424.224,174.230,25.060,154.362
C01527=1076.982,182.171,424.246,174.228,25.057,154.361
C01528=1076.977,181.922,424.269,174.225,25.054,154.361
C01529=1076.971,181.672,424.291,174.224,25.052,154.361
C01530=1076.965,181.424,424.314,174.221,25.050,154.361
C01531=1076.960,181.175,424.337,174.219,25.047,154.360
C01532=1076.954,180.927,424.359,174.217,25.045,154.360
C01533=1076.948,180.677,424.381,174.215,25.042,154.360
C01534=1076.943,180.428,424.404,174.213,25.040,154.360
C01535=1076.937,180.179,424.427,174.211,25.037,154.359
C01536=1076.931,179.930,424.449,174.208,25.035,154.359
C01537=1076.925,179.681,424.472,174.207,25.032,154.359
C01538=1076.920,179.433,424.495,174.204,25.030,154.359
C01539=1076.915,179.184,424.517,174.202,25.027,154.358
C01540=1076.908,178.935,424.539,174.200,25.025,154.358
C01541=1076.902,178.686,424.562,174.198,25.023,154.358
C01542=1076.897,178.437,424.584,174.196,25.020,154.358
C01543=1076.890,178.188,424.607,174.194,25.017,154.357
C01544=1076.886,177.939,424.629,174.191,25.015,154.357
C01545=1076.880,177.690,424.651,174.190,25.013,154.357
C01546=1076.874,177.441,424.674,174.187,25.010,154.357
C01547=1076.868,177.192,424.696,174.185,25.008,154.356
C01548=1076.862,176.943,424.719,174.183,25.005,154.356
C01549=1076.857,176.695,424.741,174.181,25.003,154.356
C01550=1076.851,176.446,424.763,174.179,25.000,154.356
C01551=1076.846,176.196,424.785,174.176,24.998,154.356
C01552=1076.840,175.948,424.808,174.174,24.995,154.355
C01553=1076.834,175.666,424.833,174.172,24.993,154.355
C01554=1076.828,175.386,424.858,174.170,24.990,154.355
C01555=1076.821,175.106,424.883,174.167,24.987,154.354
C01556=1076.814,174.825,424.908,174.165,24.984,154.354
C01557=1076.809,174.575,424.931,174.163,24.982,154.354
C01558=1076.803,174.326,424.954,174.161,24.979,154.354
C01559=1076.798,174.078,424.975,174.159,24.977,154.353
C01560=1076.792,173.828,424.997,174.156,24.974,154.353
C01561=1076.786,173.580,425.020,174.155,24.972,154.353
C01562=1076.781,173.331,425.041,174.153,24.970,154.353
C01563=1076.775,173.082,425.064,174.150,24.967,154.352
C01564=1076.770,172.833,425.086,174.148,24.964,154.352
C01565=1076.763,172.583,425.108,174.147,24.962,154.352
C01566=1076.758,172.335,425.131,174.144,24.959,154.351
C01567=1076.752,172.086,425.152,174.142,24.957,154.351
C01568=1076.747,171.837,425.175,174.140,24.954,154.351
C01569=1076.742,171.588,425.197,174.138,24.952,154.351
C01570=1076.735,171.339,425.219,174.136,24.949,154.350
C01571=1076.731,171.090,425.241,174.134,24.947,154.350
C01572=1076.725,170.841,425.264,174.132,24.945,154.350
C01573=1076.719,170.592,425.285,174.130,24.942,154.350
C01574=1076.714,170.343,425.307,174.128,24.940,154.349
C01575=1076.708,170.094,425.329,174.126,24.937,154.349
C01576=1076.702,169.845,425.352,174.124,24.934,154.349
C01577=1076.697,169.596,425.373,174.121,24.932,154.349
C01578=1076.691,169.347,425.395,174.120,24.929,154.348
C01579=1076.686,169.098,425.417,174.117,24.927,154.348
C01580=1076.680,168.850,425.439,174.115,24.924,154.348
C01581=1076.674,168.600,425.462,174.114,24.922,154.348
C01582=1076.669,168.352,425.483,174.111,24.919,154.347
C01583=1076.663,168.102,425.505,174.109,24.916,154.347
C01584=1076.659,167.854,425.527,174.108,24.915,154.347
C01585=1076.652,167.605,425.549,174.105,24.912,154.347
C01586=1076.647,167.356,425.571,174.103,24.909,154.346
C01587=1076.641,167.107,425.593,174.101,24.907,154.346
C01588=1076.636,166.857,425.615,174.099,24.904,154.346
C01589=1076.630,166.609,425.636,174.097,24.902,154.345
C01590=1076.625,166.359,425.659,174.095,24.899,154.345
C01591=1076.620,166.111,425.680,174.093,24.897,154.345
C01592=1076.614,165.861,425.702,174.092,24.894,154.345
C01593=1076.609,165.613,425.724,174.089,24.892,154.344
C01594=1076.602,165.364,425.746,174.087,24.889,154.344
C01595=1076.598,165.115,425.768,174.086,24.887,154.344
C01596=1076.591,164.866,425.790,174.083,24.884,154.344
C01597=1076.587,164.617,425.812,174.081,24.881,154.343
C01598=1076.580,164.368,425.833,174.080,24.879,154.343
C01599=1076.576,164.119,425.855,174.077,24.876,154.343
C01600=1076.569,163.870,425.877,174.075,24.874,154.342
C01601=1076.565,163.621,425.899,174.074,24.872,154.342
C01602=1076.558,163.372,425.920,174.071,24.869,154.342
C01603=1076.554,163.123,425.942,174.069,24.866,154.342
C01604=1076.548,162.875,425.963,174.067,24.864,154.341
C01605=1076.543,162.625,425.986,174.065,24.861,154.341
C01606=1076.537,162.377,426.007,174.064,24.859,154.341
C01607=1076.532,162.127,426.029,174.061,24.856,154.341
C01608=1076.526,161.879,426.050,174.059,24.854,154.340
C01609=1076.521,161.628,426.072,174.058,24.851,154.340
C01610=1076.515,161.380,426.093,174.055,24.849,154.340
C01611=1076.509,161.131,426.115,174.053,24.846,154.339
C01612=1076.504,160.882,426.137,174.052,24.844,154.339
C01613=1076.498,160.633,426.158,174.049,24.841,154.339
C01614=1076.493,160.384,426.180,174.048,24.839,154.339
C01615=1076.487,160.135,426.201,174.046,24.836,154.338
C01616=1076.482,159.886,426.223,174.043,24.834,154.338
C01617=1076.475,159.604,426.246,174.041,24.831,154.338
C01618=1076.468,159.323,426.271,174.040,24.828,154.338
C01619=1076.462,159.042,426.295,174.037,24.826,154.337
C01620=1076.456,158.762,426.319,174.035,24.823,154.337
C01621=1076.450,158.512,426.341,174.033,24.820,154.337
C01622=1076.445,158.264,426.362,174.030,24.818,154.337
C01623=1076.439,158.014,426.383,174.029,24.815,154.336
C01624=1076.433,157.765,426.405,174.027,24.813,154.336
C01625=1076.427,157.516,426.426,174.025,24.810,154.336
C01626=1076.422,157.268,426.448,174.023,24.808,154.335
C01627=1076.416,157.018,426.468,174.021,24.805,154.335
C01628=1076.411,156.769,426.490,174.019,24.803,154.335
C01629=1076.405,156.520,426.512,174.017,24.800,154.335
C01630=1076.400,156.271,426.533,174.015,24.798,154.334
C01631=1076.394,156.022,426.554,174.013,24.796,154.334
C01632=1076.388,155.773,426.575,174.012,24.793,154.334
C01633=1076.382,155.524,426.597,174.009,24.791,154.334
C01634=1076.376,155.275,426.618,174.007,24.788,154.333
C01635=1076.371,155.026,426.639,174.006,24.786,154.333
C01636=1076.366,154.777,426.660,174.003,24.783,154.333
C01637=1076.360,154.527,426.682,174.002,24.781,154.332
C01638=1076.355,154.279,426.703,173.999,24.778,154.332
C01639=1076.349,154.029,426.724,173.997,24.775,154.332
C01640=1076.343,153.781,426.745,173.996,24.773,154.332
C01641=1076.338,153.532,426.766,173.993,24.771,154.332
C01642=1076.332,153.282,426.787,173.992,24.768,154.331
C01643=1076.326,153.034,426.809,173.990,24.766,154.331
C01644=1076.320,152.784,426.830,173.988,24.763,154.331
C01645=1076.315,152.535,426.851,173.986,24.761,154.330
C01646=1076.310,152.286,426.871,173.984,24.758,154.330
C01647=1076.303,152.037,426.893,173.982,24.756,154.330
C01648=1076.298,151.788,426.914,173.980,24.753,154.330
C01649=1076.293,151.539,426.935,173.978,24.751,154.329
C01650=1076.287,151.290,426.956,173.976,24.748,154.329
C01651=1076.281,151.041,426.977,173.975,24.746,154.329
C01652=1076.276,150.792,426.998,173.972,24.744,154.329
C01653=1076.270,150.543,427.019,173.971,24.741,154.328
C01654=1076.265,150.294,427.040,173.969,24.739,154.328
C01655=1076.259,150.045,427.061,173.967,24.736,154.328
C01656=1076.253,149.795,427.082,173.965,24.734,154.328
C01657=1076.248,149.547,427.103,173.963,24.731,154.327
C01658=1076.242,149.298,427.123,173.961,24.729,154.327
C01659=1076.235,149.049,427.145,173.959,24.726,154.327
C01660=1076.230,148.800,427.165,173.957,24.724,154.326
C01661=1076.225,148.551,427.186,173.955,24.721,154.326
C01662=1076.219,148.301,427.208,173.954,24.719,154.326
C01663=1076.213,148.052,427.228,173.951,24.716,154.326
C01664=1076.208,147.804,427.249,173.950,24.714,154.325
C01665=1076.203,147.555,427.270,173.948,24.712,154.325
C01666=1076.196,147.305,427.290,173.946,24.709,154.325
C01667=1076.190,147.057,427.312,173.944,24.707,154.325
C01668=1076.185,146.808,427.332,173.943,24.704,154.324
C01669=1076.179,146.558,427.353,173.940,24.702,154.324
C01670=1076.174,146.309,427.374,173.938,24.699,154.324
C01671=1076.168,146.060,427.394,173.937,24.697,154.324
C01672=1076.162,145.811,427.415,173.934,24.694,154.323
C01673=1076.157,145.561,427.436,173.933,24.692,154.323
C01674=1076.151,145.313,427.457,173.931,24.689,154.323
C01675=1076.145,145.064,427.477,173.929,24.687,154.323
C01676=1076.139,144.814,427.498,173.927,24.684,154.322
C01677=1076.134,144.565,427.518,173.925,24.682,154.322
C01678=1076.128,144.317,427.540,173.923,24.679,154.322
C01679=1076.122,144.068,427.560,173.922,24.677,154.321
C01680=1076.117,143.818,427.581,173.919,24.674,154.321
C01681=1076.111,143.537,427.604,173.917,24.672,154.321
C01682=1076.104,143.255,427.627,173.916,24.669,154.321
C01683=1076.098,142.974,427.650,173.913,24.666,154.320
C01684=1076.092,142.693,427.673,173.911,24.663,154.320
C01685=1076.085,142.443,427.695,173.909,24.661,154.320
C01686=1076.080,142.194,427.716,173.907,24.658,154.319
C01687=1076.074,141.946,427.736,173.905,24.656,154.319
C01688=1076.069,141.696,427.756,173.904,24.653,154.319
C01689=1076.064,141.447,427.777,173.901,24.651,154.319
C01690=1076.058,141.198,427.797,173.900,24.648,154.318
C01691=1076.052,140.949,427.817,173.899,24.646,154.318
C01692=1076.047,140.700,427.838,173.896,24.643,154.318
C01693=1076.041,140.450,427.859,173.895,24.641,154.318
C01694=1076.035,140.202,427.879,173.893,24.638,154.317
C01695=1076.030,139.953,427.900,173.891,24.636,154.317
C01696=1076.023,139.704,427.920,173.889,24.633,154.317
C01697=1076.018,139.454,427.941,173.888,24.631,154.316
C01698=1076.013,139.205,427.961,173.885,24.628,154.316
C01699=1076.007,138.957,427.981,173.884,24.626,154.316
C01700=1076.001,138.707,428.002,173.882,24.623,154.316
C01701=1075.995,138.458,428.022,173.880,24.621,154.315
C01702=1075.990,138.209,428.043,173.878,24.618,154.315
C01703=1075.984,137.960,428.063,173.877,24.616,154.315
C01704=1075.978,137.711,428.083,173.874,24.613,154.315
C01705=1075.973,137.462,428.104,173.873,24.611,154.314
C01706=1075.967,137.213,428.124,173.871,24.608,154.314
C01707=1075.961,136.963,428.145,173.869,24.606,154.314
C01708=1075.955,136.714,428.165,173.867,24.604,154.314
C01709=1075.950,136.465,428.185,173.865,24.601,154.313
C01710=1075.944,136.216,428.205,173.863,24.599,154.313
C01711=1075.939,135.967,428.225,173.862,24.596,154.313
C01712=1075.933,135.718,428.245,173.859,24.594,154.312
C01713=1075.928,135.469,428.265,173.858,24.591,154.312
C01714=1075.922,135.220,428.285,173.857,24.589,154.312
C01715=1075.916,134.970,428.306,173.854,24.586,154.312
C01716=1075.910,134.721,428.326,173.853,24.584,154.311
C01717=1075.905,134.472,428.347,173.851,24.581,154.311
C01718=1075.899,134.223,428.367,173.849,24.579,154.311
C01719=1075.893,133.974,428.386,173.847,24.576,154.310
C01720=1075.888,133.725,428.407,173.846,24.574,154.310
C01721=1075.882,133.476,428.427,173.843,24.571,154.310
C01722=1075.876,133.227,428.447,173.842,24.569,154.310
C01723=1075.870,132.978,428.467,173.840,24.566,154.309
C01724=1075.865,132.729,428.488,173.838,24.564,154.309
C01725=1075.860,132.479,428.507,173.837,24.562,154.309
C01726=1075.854,132.230,428.527,173.834,24.559,154.309
C01727=1075.848,131.981,428.548,173.833,24.557,154.308
C01728=1075.842,131.732,428.568,173.831,24.554,154.308
C01729=1075.837,131.482,428.588,173.829,24.552,154.308
C01730=1075.831,131.233,428.607,173.827,24.549,154.307
C01731=1075.825,130.985,428.627,173.826,24.547,154.307
C01732=1075.819,130.736,428.647,173.823,24.544,154.307
C01733=1075.814,130.486,428.667,173.822,24.542,154.307
C01734=1075.808,130.237,428.687,173.821,24.539,154.306
C01735=1075.802,129.988,428.707,173.818,24.537,154.306
C01736=1075.796,129.738,428.727,173.817,24.534,154.306
C01737=1075.790,129.489,428.747,173.815,24.532,154.306
C01738=1075.784,129.240,428.767,173.813,24.530,154.305
C01739=1075.779,128.991,428.787,173.811,24.527,154.305
C01740=1075.773,128.742,428.806,173.809,24.525,154.305
C01741=1075.767,128.493,428.826,173.808,24.522,154.305
C01742=1075.761,128.244,428.846,173.806,24.520,154.304
C01743=1075.756,127.995,428.866,173.804,24.517,154.304
C01744=1075.750,127.745,428.885,173.802,24.515,154.304
C01745=1075.743,127.465,428.908,173.801,24.512,154.303
C01746=1075.737,127.182,428.931,173.799,24.509,154.303
C01747=1075.730,126.902,428.953,173.796,24.506,154.303
C01748=1075.723,126.620,428.975,173.794,24.503,154.302
C01749=1075.718,126.370,428.995,173.793,24.501,154.302
C01750=1075.712,126.121,429.015,173.791,24.499,154.302
C01751=1075.706,125.872,429.035,173.789,24.496,154.302
C01752=1075.701,125.623,429.054,173.788,24.494,154.301
C01753=1075.695,125.374,429.074,173.785,24.491,154.301
C01754=1075.689,125.125,429.093,173.784,24.489,154.301
C01755=1075.684,124.875,429.114,173.783,24.487,154.301
C01756=1075.678,124.626,429.133,173.780,24.483,154.300
C01757=1075.672,124.377,429.153,173.779,24.481,154.300
C01758=1075.666,124.128,429.172,173.777,24.478,154.300
C01759=1075.660,123.879,429.192,173.775,24.476,154.299
C01760=1075.655,123.630,429.211,173.773,24.473,154.299
C01761=1075.650,123.380,429.231,173.772,24.471,154.299
C01762=1075.644,123.131,429.251,173.770,24.469,154.298
C01763=1075.638,122.882,429.271,173.768,24.466,154.298
C01764=1075.633,122.633,429.290,173.767,24.463,154.298
C01765=1075.627,122.384,429.309,173.765,24.461,154.298
C01766=1075.621,122.135,429.329,173.763,24.458,154.297
C01767=1075.615,121.886,429.349,173.762,24.456,154.297
C01768=1075.610,121.636,429.368,173.759,24.453,154.297
C01769=1075.604,121.387,429.388,173.758,24.451,154.297
C01770=1075.599,121.138,429.408,173.757,24.449,154.296
C01771=1075.593,120.888,429.427,173.754,24.446,154.296
C01772=1075.587,120.640,429.447,173.753,24.444,154.296
C01773=1075.581,120.390,429.466,173.751,24.441,154.295
C01774=1075.575,120.141,429.486,173.749,24.439,154.295
C01775=1075.570,119.893,429.505,173.748,24.436,154.295
C01776=1075.565,119.643,429.524,173.746,24.433,154.295
C01777=1075.559,119.394,429.543,173.744,24.431,154.294
C01778=1075.553,119.145,429.563,173.742,24.428,154.294
C01779=1075.548,118.895,429.583,173.741,24.426,154.294
C01780=1075.542,118.646,429.602,173.739,24.423,154.293
C01781=1075.536,118.397,429.622,173.737,24.421,154.293
C01782=1075.531,118.148,429.641,173.736,24.418,154.293
C01783=1075.525,117.899,429.660,173.734,24.416,154.293
C01784=1075.520,117.649,429.680,173.732,24.413,154.292
C01785=1075.514,117.400,429.700,173.731,24.410,154.292
C01786=1075.508,117.151,429.719,173.729,24.408,154.292
C01787=1075.502,116.902,429.738,173.727,24.405,154.291
C01788=1075.497,116.653,429.757,173.726,24.403,154.291
C01789=1075.492,116.403,429.776,173.724,24.400,154.291
C01790=1075.486,116.155,429.796,173.722,24.398,154.290
C01791=1075.480,115.905,429.815,173.721,24.395,154.290
C01792=1075.474,115.656,429.835,173.719,24.392,154.290
C01793=1075.469,115.407,429.854,173.717,24.390,154.290
C01794=1075.463,115.158,429.873,173.716,24.388,154.289
C01795=1075.457,114.909,429.893,173.714,24.385,154.289
C01796=1075.452,114.659,429.912,173.712,24.383,154.289
C01797=1075.447,114.410,429.932,173.711,24.380,154.288
C01798=1075.441,114.161,429.950,173.709,24.377,154.288
C01799=1075.435,113.912,429.969,173.707,24.375,154.288
C01800=1075.430,113.662,429.989,173.705,24.372,154.287
C01801=1075.424,113.413,430.008,173.704,24.370,154.287
C01802=1075.418,113.163,430.027,173.702,24.367,154.287
C01803=1075.413,112.915,430.046,173.700,24.364,154.287
C01804=1075.407,112.666,430.065,173.699,24.362,154.286
C01805=1075.401,112.416,430.084,173.697,24.360,154.286
C01806=1075.395,112.167,430.104,173.695,24.357,154.286
C01807=1075.389,111.918,430.123,173.694,24.355,154.285
C01808=1075.384,111.669,430.142,173.693,24.352,154.285
C01809=1075.378,111.387,430.163,173.690,24.349,154.285
